LIN {X 0,Y 523.987,Z 450.894,A -85,B 0,C 180,E1 -4780.823,E2 -4780.823} C_VEL
LIN {X 0,Y 524.213,Z 441.663,A -85,B 0,C 180,E1 -4782.19,E2 -4782.19} C_VEL
LIN {X 0,Y 524.572,Z 432.281,A -85,B 0,C 180,E1 -4783.362,E2 -4783.362} C_VEL
LIN {X 0,Y 525.021,Z 420.113,A -85,B 0,C 180,E1 -4784.635,E2 -4784.635} C_VEL
LIN {X 0,Y 525.435,Z 408.795,A -85,B 0,C 180,E1 -4785.626,E2 -4785.626} C_VEL
LIN {X 0,Y 525.945,Z 395.479,A -85,B 0,C 180,E1 -4786.596,E2 -4786.596} C_VEL
LIN {X 0,Y 526.353,Z 382.284,A -85,B 0,C 180,E1 -4787.383,E2 -4787.383} C_VEL
LIN {X 0,Y 526.835,Z 368.983,A -85,B 0,C 180,E1 -4788.018,E2 -4788.018} C_VEL
LIN {X 0,Y 527.198,Z 354.45,A -85,B 0,C 180,E1 -4788.559,E2 -4788.559} C_VEL
LIN {X 0,Y 527.465,Z 339.899,A -85,B 0,C 180,E1 -4788.947,E2 -4788.947} C_VEL
LIN {X 0,Y 527.698,Z 319.361,A -85,B 0,C 180,E1 -4789.281,E2 -4789.281} C_VEL
LIN {X 0,Y 528.518,Z 183.704,A -85,B 0,C 180,E1 -4791.174,E2 -4791.174} C_VEL
LIN {X 0,Y 525.728,Z 169.853,A -85,B 0,C 180,E1 -4791.514,E2 -4791.514} C_VEL
LIN {X 0,Y 526.312,Z 151.353,A -85,B 0,C 180,E1 -4794.034,E2 -4794.034} C_VEL
LIN {X 0,Y 526.522,Z 142.38,A -85,B 0,C 180,E1 -4795.286,E2 -4795.286} C_VEL
LIN {X 0,Y 524.011,Z 130.952,A -85,B 0,C 180,E1 -4797.076,E2 -4797.076} C_VEL
LIN {X 0,Y 523.943,Z 130.846,A -85,B 0,C 180,E1 -4799.756,E2 -4799.756} C_VEL
LIN {X 0,Y 523.934,Z 130.835,A -85,B 0,C 180,E1 -4802.45,E2 -4802.45} C_VEL
LIN {X 0,Y 523.92,Z 130.845,A -85,B 0,C 180,E1 -4805.227,E2 -4805.227} C_VEL
LIN {X 0,Y 523.917,Z 130.849,A -85,B 0,C 180,E1 -4808.102,E2 -4808.102} C_VEL
LIN {X 0,Y 523.939,Z 130.842,A -85,B 0,C 180,E1 -4811.092,E2 -4811.092} C_VEL
LIN {X 0,Y 523.932,Z 130.842,A -85,B 0,C 180,E1 -4814.229,E2 -4814.229} C_VEL
LIN {X 0,Y 523.922,Z 130.844,A -85,B 0,C 180,E1 -4816.833,E2 -4816.833} C_VEL
LIN {X 0,Y 523.938,Z 130.839,A -85,B 0,C 180,E1 -4819.87,E2 -4819.87} C_VEL
LIN {X 0,Y 523.908,Z 130.847,A -85,B 0,C 180,E1 -4822.868,E2 -4822.868} C_VEL
LIN {X 0,Y 523.921,Z 130.836,A -85,B 0,C 180,E1 -4825.709,E2 -4825.709} C_VEL
LIN {X 0,Y 523.92,Z 130.835,A -85,B 0,C 180,E1 -4828.456,E2 -4828.456} C_VEL
LIN {X 0,Y 523.936,Z 130.847,A -85,B 0,C 180,E1 -4831.125,E2 -4831.125} C_VEL
LIN {X 0,Y 523.984,Z 130.833,A -85,B 0,C 180,E1 -4833.981,E2 -4833.981} C_VEL
LIN {X 0,Y 523.925,Z 130.843,A -85,B 0,C 180,E1 -4836.27,E2 -4836.27} C_VEL
LIN {X 0,Y 523.947,Z 130.842,A -85,B 0,C 180,E1 -4838.767,E2 -4838.767} C_VEL
LIN {X 0,Y 523.939,Z 130.847,A -85,B 0,C 180,E1 -4841.22,E2 -4841.22} C_VEL
LIN {X 0,Y 523.923,Z 130.84,A -85,B 0,C 180,E1 -4843.639,E2 -4843.639} C_VEL
LIN {X 0,Y 523.933,Z 130.841,A -85,B 0,C 180,E1 -4846.028,E2 -4846.028} C_VEL
LIN {X 0,Y 524.015,Z 130.835,A -85,B 0,C 180,E1 -4848.394,E2 -4848.394} C_VEL
LIN {X 0,Y 523.989,Z 130.833,A -85,B 0,C 180,E1 -4851.516,E2 -4851.516} C_VEL
LIN {X 0,Y 524.079,Z 130.829,A -85,B 0,C 180,E1 -4854.614,E2 -4854.614} C_VEL
LIN {X 0,Y 524.112,Z 130.817,A -85,B 0,C 180,E1 -4857.695,E2 -4857.695} C_VEL
LIN {X 0,Y 524.122,Z 130.819,A -85,B 0,C 180,E1 -4860.768,E2 -4860.768} C_VEL
LIN {X 0,Y 524.032,Z 130.827,A -85,B 0,C 180,E1 -4863.075,E2 -4863.075} C_VEL
LIN {X 0,Y 524.029,Z 130.837,A -85,B 0,C 180,E1 -4866.159,E2 -4866.159} C_VEL
LIN {X 0,Y 523.987,Z 130.831,A -85,B 0,C 180,E1 -4869.262,E2 -4869.262} C_VEL
LIN {X 0,Y 524.001,Z 130.837,A -85,B 0,C 180,E1 -4871.737,E2 -4871.737} C_VEL
LIN {X 0,Y 523.989,Z 130.831,A -85,B 0,C 180,E1 -4875.049,E2 -4875.049} C_VEL
LIN {X 0,Y 523.916,Z 130.852,A -85,B 0,C 180,E1 -4877.971,E2 -4877.971} C_VEL
LIN {X 0,Y 523.959,Z 130.839,A -85,B 0,C 180,E1 -4880.411,E2 -4880.411} C_VEL
LIN {X 0,Y 523.908,Z 130.845,A -85,B 0,C 180,E1 -4882.894,E2 -4882.894} C_VEL
LIN {X 0,Y 523.901,Z 130.846,A -85,B 0,C 180,E1 -4885.421,E2 -4885.421} C_VEL
LIN {X 0,Y 523.912,Z 130.849,A -85,B 0,C 180,E1 -4888.002,E2 -4888.002} C_VEL
LIN {X 0,Y 523.936,Z 130.835,A -85,B 0,C 180,E1 -4890.853,E2 -4890.853} C_VEL
LIN {X 0,Y 523.927,Z 130.841,A -85,B 0,C 180,E1 -4893.729,E2 -4893.729} C_VEL
LIN {X 0,Y 523.898,Z 130.847,A -85,B 0,C 180,E1 -4896.4,E2 -4896.4} C_VEL
LIN {X 0,Y 523.912,Z 130.845,A -85,B 0,C 180,E1 -4899.086,E2 -4899.086} C_VEL
LIN {X 0,Y 523.899,Z 130.845,A -85,B 0,C 180,E1 -4902.124,E2 -4902.124} C_VEL
LIN {X 0,Y 523.934,Z 130.842,A -85,B 0,C 180,E1 -4905.311,E2 -4905.311} C_VEL
LIN {X 0,Y 523.878,Z 130.847,A -85,B 0,C 180,E1 -4906.896,E2 -4906.896} C_VEL
LIN {X 0,Y 523.2,Z 130.938,A -85,B 0,C 180,E1 -4907.538,E2 -4907.538} C_VEL
LIN {X 0,Y 520.357,Z 131.291,A -85,B 0,C 180,E1 -4908.579,E2 -4908.579} C_VEL
LIN {X 0,Y 517.964,Z 131.586,A -85,B 0,C 180,E1 -4909.418,E2 -4909.418} C_VEL
LIN {X 0,Y 516.94,Z 131.709,A -85,B 0,C 180,E1 -4910.066,E2 -4910.066} C_VEL
LIN {X 0,Y 516.858,Z 131.719,A -85,B 0,C 180,E1 -4910.285,E2 -4910.285} C_VEL
LIN {X 0,Y 516.85,Z 131.726,A -85,B 0,C 180,E1 -4913.252,E2 -4913.252} C_VEL
LIN {X 0,Y 516.879,Z 131.722,A -85,B 0,C 180,E1 -4916.118,E2 -4916.118} C_VEL
LIN {X 0,Y 516.849,Z 131.72,A -85,B 0,C 180,E1 -4918.944,E2 -4918.944} C_VEL
LIN {X 0,Y 516.856,Z 131.728,A -85,B 0,C 180,E1 -4922.11,E2 -4922.11} C_VEL
LIN {X 0,Y 516.864,Z 131.779,A -85,B 0,C 180,E1 -4923.695,E2 -4923.695} C_VEL
LIN {X 0,Y 517.122,Z 133.046,A -85,B 0,C 180,E1 -4923.969,E2 -4923.969} C_VEL
LIN {X 0,Y 519.393,Z 143.168,A -85,B 0,C 180,E1 -4925.625,E2 -4925.625} C_VEL
LIN {X 0,Y 519.177,Z 153.314,A -85,B 0,C 180,E1 -4927.13,E2 -4927.13} C_VEL
LIN {X 0,Y 518.951,Z 161.322,A -85,B 0,C 180,E1 -4928.255,E2 -4928.255} C_VEL
LIN {X 0,Y 521.967,Z 176.108,A -85,B 0,C 180,E1 -4928.615,E2 -4928.615} C_VEL
LIN {X 0,Y 520.906,Z 326.105,A -85,B 0,C 180,E1 -4930.75,E2 -4930.75} C_VEL
LIN {X 0,Y 520.589,Z 341.471,A -85,B 0,C 180,E1 -4931.12,E2 -4931.12} C_VEL
LIN {X 0,Y 520.263,Z 356.352,A -85,B 0,C 180,E1 -4931.644,E2 -4931.644} C_VEL
LIN {X 0,Y 519.75,Z 370.274,A -85,B 0,C 180,E1 -4932.287,E2 -4932.287} C_VEL
LIN {X 0,Y 519.241,Z 383.909,A -85,B 0,C 180,E1 -4933.082,E2 -4933.082} C_VEL
LIN {X 0,Y 518.727,Z 396.578,A -85,B 0,C 180,E1 -4933.986,E2 -4933.986} C_VEL
LIN {X 0,Y 518.184,Z 409.14,A -85,B 0,C 180,E1 -4935.067,E2 -4935.067} C_VEL
LIN {X 0,Y 517.708,Z 420.65,A -85,B 0,C 180,E1 -4936.257,E2 -4936.257} C_VEL
LIN {X 0,Y 517.314,Z 430.339,A -85,B 0,C 180,E1 -4937.445,E2 -4937.445} C_VEL
LIN {X 0,Y 517.023,Z 439.835,A -85,B 0,C 180,E1 -4938.831,E2 -4938.831} C_VEL
LIN {X 0,Y 516.725,Z 447.744,A -85,B 0,C 180,E1 -4940.211,E2 -4940.211} C_VEL
LIN {X 0,Y 516.511,Z 455.13,A -85,B 0,C 180,E1 -4941.786,E2 -4941.786} C_VEL
LIN {X 0,Y 516.394,Z 459.661,A -85,B 0,C 180,E1 -4942.964,E2 -4942.964} C_VEL
LIN {X 0,Y 516.379,Z 464.465,A -85,B 0,C 180,E1 -4944.533,E2 -4944.533} C_VEL
LIN {X 0,Y 516.307,Z 467.988,A -85,B 0,C 180,E1 -4946.097,E2 -4946.097} C_VEL
LIN {X 0,Y 516.259,Z 470.322,A -85,B 0,C 180,E1 -4947.659,E2 -4947.659} C_VEL
LIN {X 0,Y 516.156,Z 471.518,A -85,B 0,C 180,E1 -4949.22,E2 -4949.22} C_VEL
LIN {X 0,Y 516.157,Z 471.537,A -85,B 0,C 180,E1 -4950.78,E2 -4950.78} C_VEL
LIN {X 0,Y 516.259,Z 470.418,A -85,B 0,C 180,E1 -4952.341,E2 -4952.341} C_VEL
LIN {X 0,Y 516.308,Z 468.16,A -85,B 0,C 180,E1 -4953.903,E2 -4953.903} C_VEL
LIN {X 0,Y 516.374,Z 464.708,A -85,B 0,C 180,E1 -4955.467,E2 -4955.467} C_VEL
LIN {X 0,Y 516.393,Z 459.982,A -85,B 0,C 180,E1 -4957.036,E2 -4957.036} C_VEL
LIN {X 0,Y 516.542,Z 453.859,A -85,B 0,C 180,E1 -4958.608,E2 -4958.608} C_VEL
LIN {X 0,Y 516.767,Z 446.151,A -85,B 0,C 180,E1 -4960.183,E2 -4960.183} C_VEL
LIN {X 0,Y 517.008,Z 437.932,A -85,B 0,C 180,E1 -4961.567,E2 -4961.567} C_VEL
LIN {X 0,Y 517.394,Z 428.037,A -85,B 0,C 180,E1 -4962.952,E2 -4962.952} C_VEL
LIN {X 0,Y 517.838,Z 417.892,A -85,B 0,C 180,E1 -4964.14,E2 -4964.14} C_VEL
LIN {X 0,Y 518.342,Z 406.115,A -85,B 0,C 180,E1 -4965.303,E2 -4965.303} C_VEL
LIN {X 0,Y 518.84,Z 393.976,A -85,B 0,C 180,E1 -4966.304,E2 -4966.304} C_VEL
LIN {X 0,Y 519.399,Z 380.576,A -85,B 0,C 180,E1 -4967.217,E2 -4967.217} C_VEL
LIN {X 0,Y 519.804,Z 368.066,A -85,B 0,C 180,E1 -4967.914,E2 -4967.914} C_VEL
LIN {X 0,Y 520.338,Z 353.435,A -85,B 0,C 180,E1 -4968.557,E2 -4968.557} C_VEL
LIN {X 0,Y 520.652,Z 338.696,A -85,B 0,C 180,E1 -4969.044,E2 -4969.044} C_VEL
LIN {X 0,Y 520.941,Z 323.655,A -85,B 0,C 180,E1 -4969.38,E2 -4969.38} C_VEL
LIN {X 0,Y 522.001,Z 175.538,A -85,B 0,C 180,E1 -4971.482,E2 -4971.482} C_VEL
LIN {X 0,Y 518.92,Z 161.155,A -85,B 0,C 180,E1 -4971.846,E2 -4971.846} C_VEL
LIN {X 0,Y 519.489,Z 145.188,A -85,B 0,C 180,E1 -4974.157,E2 -4974.157} C_VEL
LIN {X 0,Y 518.911,Z 140.798,A -85,B 0,C 180,E1 -4974.847,E2 -4974.847} C_VEL
LIN {X 0,Y 516.893,Z 132.05,A -85,B 0,C 180,E1 -4976.307,E2 -4976.307} C_VEL
LIN {X 0,Y 516.828,Z 131.719,A -85,B 0,C 180,E1 -4976.663,E2 -4976.663} C_VEL
LIN {X 0,Y 516.838,Z 131.719,A -85,B 0,C 180,E1 -4979.509,E2 -4979.509} C_VEL
LIN {X 0,Y 516.867,Z 131.726,A -85,B 0,C 180,E1 -4982.538,E2 -4982.538} C_VEL
LIN {X 0,Y 516.851,Z 131.729,A -85,B 0,C 180,E1 -4985.327,E2 -4985.327} C_VEL
LIN {X 0,Y 516.869,Z 131.728,A -85,B 0,C 180,E1 -4988.717,E2 -4988.717} C_VEL
LIN {X 0,Y 516.845,Z 131.726,A -85,B 0,C 180,E1 -4991.782,E2 -4991.782} C_VEL
LIN {X 0,Y 516.897,Z 131.722,A -85,B 0,C 180,E1 -4995.007,E2 -4995.007} C_VEL
LIN {X 0,Y 516.85,Z 131.728,A -85,B 0,C 180,E1 -4998.407,E2 -4998.407} C_VEL
LIN {X 0,Y 516.875,Z 131.719,A -85,B 0,C 180,E1 -5001.283,E2 -5001.283} C_VEL
LIN {X 0,Y 516.866,Z 131.727,A -85,B 0,C 180,E1 -5004.219,E2 -5004.219} C_VEL
LIN {X 0,Y 516.882,Z 131.707,A -85,B 0,C 180,E1 -5007.052,E2 -5007.052} C_VEL
LIN {X 0,Y 516.866,Z 131.715,A -85,B 0,C 180,E1 -5009.795,E2 -5009.795} C_VEL
LIN {X 0,Y 516.876,Z 131.728,A -85,B 0,C 180,E1 -5012.464,E2 -5012.464} C_VEL
LIN {X 0,Y 516.847,Z 131.721,A -85,B 0,C 180,E1 -5015.068,E2 -5015.068} C_VEL
LIN {X 0,Y 516.871,Z 131.724,A -85,B 0,C 180,E1 -5017.622,E2 -5017.622} C_VEL
LIN {X 0,Y 516.92,Z 131.718,A -85,B 0,C 180,E1 -5020.129,E2 -5020.129} C_VEL
LIN {X 0,Y 516.881,Z 131.723,A -85,B 0,C 180,E1 -5022.594,E2 -5022.594} C_VEL
LIN {X 0,Y 516.938,Z 131.709,A -85,B 0,C 180,E1 -5025.03,E2 -5025.03} C_VEL
LIN {X 0,Y 516.969,Z 131.714,A -85,B 0,C 180,E1 -5028.234,E2 -5028.234} C_VEL
LIN {X 0,Y 516.955,Z 131.711,A -85,B 0,C 180,E1 -5031.399,E2 -5031.399} C_VEL
LIN {X 0,Y 517.022,Z 131.703,A -85,B 0,C 180,E1 -5034.54,E2 -5034.54} C_VEL
LIN {X 0,Y 517.081,Z 131.696,A -85,B 0,C 180,E1 -5037.663,E2 -5037.663} C_VEL
LIN {X 0,Y 517.088,Z 131.697,A -85,B 0,C 180,E1 -5040,E2 -5040} C_VEL
LIN {X 0,Y 517.082,Z 131.692,A -85,B 0,C 180,E1 -5042.337,E2 -5042.337} C_VEL
LIN {X 0,Y 517.025,Z 131.708,A -85,B 0,C 180,E1 -5045.46,E2 -5045.46} C_VEL
LIN {X 0,Y 516.957,Z 131.709,A -85,B 0,C 180,E1 -5048.6,E2 -5048.6} C_VEL
LIN {X 0,Y 516.954,Z 131.713,A -85,B 0,C 180,E1 -5051.807,E2 -5051.807} C_VEL
LIN {X 0,Y 516.945,Z 131.714,A -85,B 0,C 180,E1 -5055.145,E2 -5055.145} C_VEL
LIN {X 0,Y 516.914,Z 131.717,A -85,B 0,C 180,E1 -5058.223,E2 -5058.223} C_VEL
LIN {X 0,Y 516.914,Z 131.719,A -85,B 0,C 180,E1 -5060.701,E2 -5060.701} C_VEL
LIN {X 0,Y 516.887,Z 131.72,A -85,B 0,C 180,E1 -5064.073,E2 -5064.073} C_VEL
LIN {X 0,Y 516.91,Z 131.719,A -85,B 0,C 180,E1 -5066.659,E2 -5066.659} C_VEL
LIN {X 0,Y 516.911,Z 131.716,A -85,B 0,C 180,E1 -5069.523,E2 -5069.523} C_VEL
LIN {X 0,Y 516.895,Z 131.708,A -85,B 0,C 180,E1 -5072.543,E2 -5072.543} C_VEL
LIN {X 0,Y 516.867,Z 131.721,A -85,B 0,C 180,E1 -5075.329,E2 -5075.329} C_VEL
LIN {X 0,Y 516.881,Z 131.723,A -85,B 0,C 180,E1 -5077.943,E2 -5077.943} C_VEL
LIN {X 0,Y 516.884,Z 131.717,A -85,B 0,C 180,E1 -5080.742,E2 -5080.742} C_VEL
LIN {X 0,Y 516.885,Z 131.723,A -85,B 0,C 180,E1 -5082.831,E2 -5082.831} C_VEL
LIN {X 0,Y 516.896,Z 131.715,A -85,B 0,C 180,E1 -5085.007,E2 -5085.007} C_VEL
LIN {X 0,Y 516.914,Z 131.722,A -85,B 0,C 180,E1 -5088.399,E2 -5088.399} C_VEL
LIN {X 0,Y 516.883,Z 131.719,A -85,B 0,C 180,E1 -5091.284,E2 -5091.284} C_VEL
LIN {X 0,Y 516.872,Z 131.724,A -85,B 0,C 180,E1 -5094.22,E2 -5094.22} C_VEL
LIN {X 0,Y 516.895,Z 131.715,A -85,B 0,C 180,E1 -5097.053,E2 -5097.053} C_VEL
LIN {X 0,Y 516.893,Z 131.723,A -85,B 0,C 180,E1 -5099.796,E2 -5099.796} C_VEL
LIN {X 0,Y 516.941,Z 131.828,A -85,B 0,C 180,E1 -5102.66,E2 -5102.66} C_VEL
LIN {X 0,Y 519.647,Z 143.76,A -85,B 0,C 180,E1 -5104.562,E2 -5104.562} C_VEL
LIN {X 0,Y 519.417,Z 154.273,A -85,B 0,C 180,E1 -5106.051,E2 -5106.051} C_VEL
LIN {X 0,Y 518.893,Z 169.735,A -85,B 0,C 180,E1 -5108.185,E2 -5108.185} C_VEL
LIN {X 0,Y 521.944,Z 185.319,A -85,B 0,C 180,E1 -5108.571,E2 -5108.571} C_VEL
LIN {X 0,Y 520.888,Z 335.251,A -85,B 0,C 180,E1 -5110.704,E2 -5110.704} C_VEL
LIN {X 0,Y 520.559,Z 350.405,A -85,B 0,C 180,E1 -5111.067,E2 -5111.067} C_VEL
LIN {X 0,Y 520.171,Z 365.412,A -85,B 0,C 180,E1 -5111.59,E2 -5111.59} C_VEL
LIN {X 0,Y 519.646,Z 380.411,A -85,B 0,C 180,E1 -5112.284,E2 -5112.284} C_VEL
LIN {X 0,Y 519.132,Z 393.896,A -85,B 0,C 180,E1 -5113.078,E2 -5113.078} C_VEL
LIN {X 0,Y 518.614,Z 407.626,A -85,B 0,C 180,E1 -5114.073,E2 -5114.073} C_VEL
LIN {X 0,Y 518.057,Z 420.039,A -85,B 0,C 180,E1 -5115.164,E2 -5115.164} C_VEL
LIN {X 0,Y 517.593,Z 432.215,A -85,B 0,C 180,E1 -5116.454,E2 -5116.454} C_VEL
LIN {X 0,Y 517.146,Z 443.038,A -85,B 0,C 180,E1 -5117.84,E2 -5117.84} C_VEL
LIN {X 0,Y 516.895,Z 452.046,A -85,B 0,C 180,E1 -5119.225,E2 -5119.225} C_VEL
LIN {X 0,Y 516.601,Z 459.516,A -85,B 0,C 180,E1 -5120.604,E2 -5120.604} C_VEL
LIN {X 0,Y 516.451,Z 466.485,A -85,B 0,C 180,E1 -5122.179,E2 -5122.179} C_VEL
LIN {X 0,Y 516.36,Z 471.963,A -85,B 0,C 180,E1 -5123.749,E2 -5123.749} C_VEL
LIN {X 0,Y 516.239,Z 476.102,A -85,B 0,C 180,E1 -5125.315,E2 -5125.315} C_VEL
LIN {X 0,Y 516.27,Z 479.005,A -85,B 0,C 180,E1 -5126.879,E2 -5126.879} C_VEL
LIN {X 0,Y 516.189,Z 480.735,A -85,B 0,C 180,E1 -5128.44,E2 -5128.44} C_VEL
LIN {X 0,Y 516.151,Z 481.328,A -85,B 0,C 180,E1 -5130,E2 -5130} C_VEL
LIN {X 0,Y 516.189,Z 480.733,A -85,B 0,C 180,E1 -5131.56,E2 -5131.56} C_VEL
LIN {X 0,Y 516.27,Z 479,A -85,B 0,C 180,E1 -5133.121,E2 -5133.121} C_VEL
LIN {X 0,Y 516.239,Z 476.1,A -85,B 0,C 180,E1 -5134.685,E2 -5134.685} C_VEL
LIN {X 0,Y 516.376,Z 471.967,A -85,B 0,C 180,E1 -5136.251,E2 -5136.251} C_VEL
LIN {X 0,Y 516.451,Z 466.486,A -85,B 0,C 180,E1 -5137.821,E2 -5137.821} C_VEL
LIN {X 0,Y 516.601,Z 459.51,A -85,B 0,C 180,E1 -5139.396,E2 -5139.396} C_VEL
LIN {X 0,Y 516.952,Z 450.827,A -85,B 0,C 180,E1 -5140.972,E2 -5140.972} C_VEL
LIN {X 0,Y 517.202,Z 441.748,A -85,B 0,C 180,E1 -5142.338,E2 -5142.338} C_VEL
LIN {X 0,Y 517.593,Z 432.214,A -85,B 0,C 180,E1 -5143.546,E2 -5143.546} C_VEL
LIN {X 0,Y 518.092,Z 420.046,A -85,B 0,C 180,E1 -5144.835,E2 -5144.835} C_VEL
LIN {X 0,Y 518.59,Z 407.889,A -85,B 0,C 180,E1 -5145.908,E2 -5145.908} C_VEL
LIN {X 0,Y 519.082,Z 395.412,A -85,B 0,C 180,E1 -5146.822,E2 -5146.822} C_VEL
LIN {X 0,Y 519.543,Z 382.217,A -85,B 0,C 180,E1 -5147.618,E2 -5147.618} C_VEL
LIN {X 0,Y 520.123,Z 367.788,A -85,B 0,C 180,E1 -5148.31,E2 -5148.31} C_VEL
LIN {X 0,Y 520.471,Z 353.62,A -85,B 0,C 180,E1 -5148.833,E2 -5148.833} C_VEL
LIN {X 0,Y 520.812,Z 338.587,A -85,B 0,C 180,E1 -5149.227,E2 -5149.227} C_VEL
LIN {X 0,Y 521.012,Z 316.274,A -85,B 0,C 180,E1 -5149.582,E2 -5149.582} C_VEL
LIN {X 0,Y 521.92,Z 184.769,A -85,B 0,C 180,E1 -5151.438,E2 -5151.438} C_VEL
LIN {X 0,Y 518.869,Z 169.838,A -85,B 0,C 180,E1 -5151.809,E2 -5151.809} C_VEL
LIN {X 0,Y 519.47,Z 152.785,A -85,B 0,C 180,E1 -5154.158,E2 -5154.158} C_VEL
LIN {X 0,Y 519.759,Z 144.939,A -85,B 0,C 180,E1 -5155.263,E2 -5155.263} C_VEL
LIN {X 0,Y 517.664,Z 134.82,A -85,B 0,C 180,E1 -5156.834,E2 -5156.834} C_VEL
LIN {X 0,Y 516.957,Z 131.788,A -85,B 0,C 180,E1 -5157.366,E2 -5157.366} C_VEL
LIN {X 0,Y 516.893,Z 131.723,A -85,B 0,C 180,E1 -5160.204,E2 -5160.204} C_VEL
LIN {X 0,Y 516.895,Z 131.716,A -85,B 0,C 180,E1 -5162.947,E2 -5162.947} C_VEL
LIN {X 0,Y 516.871,Z 131.724,A -85,B 0,C 180,E1 -5165.78,E2 -5165.78} C_VEL
LIN {X 0,Y 516.883,Z 131.718,A -85,B 0,C 180,E1 -5168.716,E2 -5168.716} C_VEL
LIN {X 0,Y 516.912,Z 131.725,A -85,B 0,C 180,E1 -5171.775,E2 -5171.775} C_VEL
LIN {X 0,Y 516.895,Z 131.716,A -85,B 0,C 180,E1 -5175.007,E2 -5175.007} C_VEL
LIN {X 0,Y 516.914,Z 131.711,A -85,B 0,C 180,E1 -5178.399,E2 -5178.399} C_VEL
LIN {X 0,Y 516.881,Z 131.719,A -85,B 0,C 180,E1 -5181.284,E2 -5181.284} C_VEL
LIN {X 0,Y 516.872,Z 131.72,A -85,B 0,C 180,E1 -5184.22,E2 -5184.22} C_VEL
LIN {X 0,Y 516.882,Z 131.708,A -85,B 0,C 180,E1 -5187.052,E2 -5187.052} C_VEL
LIN {X 0,Y 516.888,Z 131.722,A -85,B 0,C 180,E1 -5189.796,E2 -5189.796} C_VEL
LIN {X 0,Y 516.926,Z 131.715,A -85,B 0,C 180,E1 -5192.467,E2 -5192.467} C_VEL
LIN {X 0,Y 516.907,Z 131.72,A -85,B 0,C 180,E1 -5195.072,E2 -5195.072} C_VEL
LIN {X 0,Y 516.887,Z 131.718,A -85,B 0,C 180,E1 -5198.462,E2 -5198.462} C_VEL
LIN {X 0,Y 516.893,Z 131.725,A -85,B 0,C 180,E1 -5200.955,E2 -5200.955} C_VEL
LIN {X 0,Y 516.899,Z 131.717,A -85,B 0,C 180,E1 -5203.41,E2 -5203.41} C_VEL
LIN {X 0,Y 516.889,Z 131.718,A -85,B 0,C 180,E1 -5205.834,E2 -5205.834} C_VEL
LIN {X 0,Y 516.952,Z 131.713,A -85,B 0,C 180,E1 -5209.028,E2 -5209.028} C_VEL
LIN {X 0,Y 516.964,Z 131.71,A -85,B 0,C 180,E1 -5212.187,E2 -5212.187} C_VEL
LIN {X 0,Y 517.026,Z 131.709,A -85,B 0,C 180,E1 -5214.54,E2 -5214.54} C_VEL
LIN {X 0,Y 517.083,Z 131.692,A -85,B 0,C 180,E1 -5217.663,E2 -5217.663} C_VEL
LIN {X 0,Y 517.092,Z 131.695,A -85,B 0,C 180,E1 -5220.779,E2 -5220.779} C_VEL
LIN {X 0,Y 516.974,Z 131.706,A -85,B 0,C 180,E1 -5223.117,E2 -5223.117} C_VEL
LIN {X 0,Y 516.991,Z 131.715,A -85,B 0,C 180,E1 -5226.243,E2 -5226.243} C_VEL
LIN {X 0,Y 516.943,Z 131.709,A -85,B 0,C 180,E1 -5229.39,E2 -5229.39} C_VEL
LIN {X 0,Y 516.954,Z 131.715,A -85,B 0,C 180,E1 -5231.807,E2 -5231.807} C_VEL
LIN {X 0,Y 516.941,Z 131.709,A -85,B 0,C 180,E1 -5235.144,E2 -5235.144} C_VEL
LIN {X 0,Y 516.879,Z 131.724,A -85,B 0,C 180,E1 -5238.224,E2 -5238.224} C_VEL
LIN {X 0,Y 516.906,Z 131.715,A -85,B 0,C 180,E1 -5240.702,E2 -5240.702} C_VEL
LIN {X 0,Y 516.886,Z 131.721,A -85,B 0,C 180,E1 -5244.073,E2 -5244.073} C_VEL
LIN {X 0,Y 516.845,Z 131.725,A -85,B 0,C 180,E1 -5246.662,E2 -5246.662} C_VEL
LIN {X 0,Y 516.887,Z 131.724,A -85,B 0,C 180,E1 -5249.519,E2 -5249.519} C_VEL
LIN {X 0,Y 516.895,Z 131.703,A -85,B 0,C 180,E1 -5252.543,E2 -5252.543} C_VEL
LIN {X 0,Y 516.861,Z 131.726,A -85,B 0,C 180,E1 -5255.329,E2 -5255.329} C_VEL
LIN {X 0,Y 516.878,Z 131.719,A -85,B 0,C 180,E1 -5257.942,E2 -5257.942} C_VEL
LIN {X 0,Y 516.853,Z 131.712,A -85,B 0,C 180,E1 -5260.745,E2 -5260.745} C_VEL
LIN {X 0,Y 516.881,Z 131.722,A -85,B 0,C 180,E1 -5263.904,E2 -5263.904} C_VEL
LIN {X 0,Y 516.836,Z 131.725,A -85,B 0,C 180,E1 -5266.896,E2 -5266.896} C_VEL
LIN {X 0,Y 516.86,Z 131.721,A -85,B 0,C 180,E1 -5269.593,E2 -5269.593} C_VEL
LIN {X 0,Y 516.858,Z 131.719,A -85,B 0,C 180,E1 -5270.285,E2 -5270.285} C_VEL
LIN {X 0,Y 516.197,Z 131.809,A -85,B 0,C 180,E1 -5270.936,E2 -5270.936} C_VEL
LIN {X 0,Y 513.348,Z 132.162,A -85,B 0,C 180,E1 -5271.991,E2 -5271.991} C_VEL
LIN {X 0,Y 510.932,Z 132.468,A -85,B 0,C 180,E1 -5272.842,E2 -5272.842} C_VEL
LIN {X 0,Y 509.888,Z 132.593,A -85,B 0,C 180,E1 -5273.498,E2 -5273.498} C_VEL
LIN {X 0,Y 509.8,Z 132.602,A -85,B 0,C 180,E1 -5273.721,E2 -5273.721} C_VEL
LIN {X 0,Y 509.839,Z 132.6,A -85,B 0,C 180,E1 -5276.538,E2 -5276.538} C_VEL
LIN {X 0,Y 509.801,Z 132.592,A -85,B 0,C 180,E1 -5279.331,E2 -5279.331} C_VEL
LIN {X 0,Y 509.823,Z 132.604,A -85,B 0,C 180,E1 -5282.05,E2 -5282.05} C_VEL
LIN {X 0,Y 509.803,Z 132.654,A -85,B 0,C 180,E1 -5283.429,E2 -5283.429} C_VEL
LIN {X 0,Y 510.265,Z 134.76,A -85,B 0,C 180,E1 -5283.849,E2 -5283.849} C_VEL
LIN {X 0,Y 512.569,Z 144.901,A -85,B 0,C 180,E1 -5285.534,E2 -5285.534} C_VEL
LIN {X 0,Y 512.234,Z 156.336,A -85,B 0,C 180,E1 -5287.247,E2 -5287.247} C_VEL
LIN {X 0,Y 512.117,Z 161.303,A -85,B 0,C 180,E1 -5287.944,E2 -5287.944} C_VEL
LIN {X 0,Y 515.308,Z 176.214,A -85,B 0,C 180,E1 -5288.324,E2 -5288.324} C_VEL
LIN {X 0,Y 514.261,Z 322.379,A -85,B 0,C 180,E1 -5290.425,E2 -5290.425} C_VEL
LIN {X 0,Y 513.998,Z 337.997,A -85,B 0,C 180,E1 -5290.768,E2 -5290.768} C_VEL
LIN {X 0,Y 513.616,Z 352.541,A -85,B 0,C 180,E1 -5291.243,E2 -5291.243} C_VEL
LIN {X 0,Y 513.103,Z 366.388,A -85,B 0,C 180,E1 -5291.844,E2 -5291.844} C_VEL
LIN {X 0,Y 512.555,Z 380.825,A -85,B 0,C 180,E1 -5292.649,E2 -5292.649} C_VEL
LIN {X 0,Y 511.971,Z 393.945,A -85,B 0,C 180,E1 -5293.553,E2 -5293.553} C_VEL
LIN {X 0,Y 511.488,Z 405.439,A -85,B 0,C 180,E1 -5294.506,E2 -5294.506} C_VEL
LIN {X 0,Y 510.948,Z 417.161,A -85,B 0,C 180,E1 -5295.665,E2 -5295.665} C_VEL
LIN {X 0,Y 510.48,Z 427.389,A -85,B 0,C 180,E1 -5296.87,E2 -5296.87} C_VEL
LIN {X 0,Y 510.051,Z 436.916,A -85,B 0,C 180,E1 -5298.201,E2 -5298.201} C_VEL
LIN {X 0,Y 509.832,Z 444.596,A -85,B 0,C 180,E1 -5299.476,E2 -5299.476} C_VEL
LIN {X 0,Y 509.551,Z 451.709,A -85,B 0,C 180,E1 -5300.874,E2 -5300.874} C_VEL
LIN {X 0,Y 509.355,Z 458.31,A -85,B 0,C 180,E1 -5302.468,E2 -5302.468} C_VEL
LIN {X 0,Y 509.304,Z 463.473,A -85,B 0,C 180,E1 -5304.06,E2 -5304.06} C_VEL
LIN {X 0,Y 509.16,Z 466.449,A -85,B 0,C 180,E1 -5305.249,E2 -5305.249} C_VEL
LIN {X 0,Y 509.188,Z 469.367,A -85,B 0,C 180,E1 -5306.835,E2 -5306.835} C_VEL
LIN {X 0,Y 509.11,Z 471.127,A -85,B 0,C 180,E1 -5308.418,E2 -5308.418} C_VEL
LIN {X 0,Y 509.064,Z 471.744,A -85,B 0,C 180,E1 -5310,E2 -5310} C_VEL
LIN {X 0,Y 509.111,Z 471.184,A -85,B 0,C 180,E1 -5311.582,E2 -5311.582} C_VEL
LIN {X 0,Y 509.189,Z 469.499,A -85,B 0,C 180,E1 -5313.165,E2 -5313.165} C_VEL
LIN {X 0,Y 509.159,Z 466.653,A -85,B 0,C 180,E1 -5314.751,E2 -5314.751} C_VEL
LIN {X 0,Y 509.287,Z 463.71,A -85,B 0,C 180,E1 -5315.941,E2 -5315.941} C_VEL
LIN {X 0,Y 509.354,Z 458.628,A -85,B 0,C 180,E1 -5317.532,E2 -5317.532} C_VEL
LIN {X 0,Y 509.544,Z 452.12,A -85,B 0,C 180,E1 -5319.127,E2 -5319.127} C_VEL
LIN {X 0,Y 509.828,Z 445.1,A -85,B 0,C 180,E1 -5320.524,E2 -5320.524} C_VEL
LIN {X 0,Y 510.081,Z 436.366,A -85,B 0,C 180,E1 -5321.971,E2 -5321.971} C_VEL
LIN {X 0,Y 510.517,Z 426.486,A -85,B 0,C 180,E1 -5323.332,E2 -5323.332} C_VEL
LIN {X 0,Y 510.979,Z 416.088,A -85,B 0,C 180,E1 -5324.537,E2 -5324.537} C_VEL
LIN {X 0,Y 511.524,Z 404.997,A -85,B 0,C 180,E1 -5325.623,E2 -5325.623} C_VEL
LIN {X 0,Y 512.062,Z 392.484,A -85,B 0,C 180,E1 -5326.649,E2 -5326.649} C_VEL
LIN {X 0,Y 512.666,Z 379.052,A -85,B 0,C 180,E1 -5327.553,E2 -5327.553} C_VEL
LIN {X 0,Y 513.217,Z 364.109,A -85,B 0,C 180,E1 -5328.359,E2 -5328.359} C_VEL
LIN {X 0,Y 513.736,Z 348.826,A -85,B 0,C 180,E1 -5328.986,E2 -5328.986} C_VEL
LIN {X 0,Y 514.063,Z 333.893,A -85,B 0,C 180,E1 -5329.433,E2 -5329.433} C_VEL
LIN {X 0,Y 514.312,Z 319.15,A -85,B 0,C 180,E1 -5329.718,E2 -5329.718} C_VEL
LIN {X 0,Y 515.386,Z 176.758,A -85,B 0,C 180,E1 -5331.754,E2 -5331.754} C_VEL
LIN {X 0,Y 512.116,Z 161.267,A -85,B 0,C 180,E1 -5332.149,E2 -5332.149} C_VEL
LIN {X 0,Y 512.657,Z 145.463,A -85,B 0,C 180,E1 -5334.467,E2 -5334.467} C_VEL
LIN {X 0,Y 509.843,Z 132.917,A -85,B 0,C 180,E1 -5336.573,E2 -5336.573} C_VEL
LIN {X 0,Y 509.782,Z 132.595,A -85,B 0,C 180,E1 -5336.771,E2 -5336.771} C_VEL
LIN {X 0,Y 509.793,Z 132.609,A -85,B 0,C 180,E1 -5338.85,E2 -5338.85} C_VEL
LIN {X 0,Y 509.789,Z 132.608,A -85,B 0,C 180,E1 -5341.592,E2 -5341.592} C_VEL
LIN {X 0,Y 509.833,Z 132.599,A -85,B 0,C 180,E1 -5344.415,E2 -5344.415} C_VEL
LIN {X 0,Y 509.783,Z 132.611,A -85,B 0,C 180,E1 -5347.344,E2 -5347.344} C_VEL
LIN {X 0,Y 509.813,Z 132.597,A -85,B 0,C 180,E1 -5350.385,E2 -5350.385} C_VEL
LIN {X 0,Y 509.806,Z 132.597,A -85,B 0,C 180,E1 -5353.573,E2 -5353.573} C_VEL
LIN {X 0,Y 509.806,Z 132.605,A -85,B 0,C 180,E1 -5356.427,E2 -5356.427} C_VEL
LIN {X 0,Y 509.813,Z 132.588,A -85,B 0,C 180,E1 -5359.615,E2 -5359.615} C_VEL
LIN {X 0,Y 509.808,Z 132.607,A -85,B 0,C 180,E1 -5362.658,E2 -5362.658} C_VEL
LIN {X 0,Y 509.84,Z 132.595,A -85,B 0,C 180,E1 -5365.801,E2 -5365.801} C_VEL
LIN {X 0,Y 509.845,Z 132.588,A -85,B 0,C 180,E1 -5368.721,E2 -5368.721} C_VEL
LIN {X 0,Y 509.838,Z 132.598,A -85,B 0,C 180,E1 -5371.153,E2 -5371.153} C_VEL
LIN {X 0,Y 509.851,Z 132.598,A -85,B 0,C 180,E1 -5373.826,E2 -5373.826} C_VEL
LIN {X 0,Y 509.82,Z 132.606,A -85,B 0,C 180,E1 -5376.436,E2 -5376.436} C_VEL
LIN {X 0,Y 509.908,Z 132.591,A -85,B 0,C 180,E1 -5379.844,E2 -5379.844} C_VEL
LIN {X 0,Y 509.854,Z 132.601,A -85,B 0,C 180,E1 -5382.347,E2 -5382.347} C_VEL
LIN {X 0,Y 509.888,Z 132.588,A -85,B 0,C 180,E1 -5384.818,E2 -5384.818} C_VEL
LIN {X 0,Y 509.904,Z 132.595,A -85,B 0,C 180,E1 -5388.124,E2 -5388.124} C_VEL
LIN {X 0,Y 509.903,Z 132.587,A -85,B 0,C 180,E1 -5391.279,E2 -5391.279} C_VEL
LIN {X 0,Y 509.973,Z 132.582,A -85,B 0,C 180,E1 -5394.464,E2 -5394.464} C_VEL
LIN {X 0,Y 510.051,Z 132.571,A -85,B 0,C 180,E1 -5397.631,E2 -5397.631} C_VEL
LIN {X 0,Y 510.02,Z 132.575,A -85,B 0,C 180,E1 -5400.789,E2 -5400.789} C_VEL
LIN {X 0,Y 509.927,Z 132.588,A -85,B 0,C 180,E1 -5403.16,E2 -5403.16} C_VEL
LIN {X 0,Y 509.943,Z 132.584,A -85,B 0,C 180,E1 -5406.33,E2 -5406.33} C_VEL
LIN {X 0,Y 509.905,Z 132.589,A -85,B 0,C 180,E1 -5408.72,E2 -5408.72} C_VEL
LIN {X 0,Y 509.907,Z 132.59,A -85,B 0,C 180,E1 -5411.932,E2 -5411.932} C_VEL
LIN {X 0,Y 509.897,Z 132.591,A -85,B 0,C 180,E1 -5415.242,E2 -5415.242} C_VEL
LIN {X 0,Y 509.859,Z 132.598,A -85,B 0,C 180,E1 -5418.484,E2 -5418.484} C_VEL
LIN {X 0,Y 509.852,Z 132.598,A -85,B 0,C 180,E1 -5421.002,E2 -5421.002} C_VEL
LIN {X 0,Y 509.821,Z 132.601,A -85,B 0,C 180,E1 -5423.564,E2 -5423.564} C_VEL
LIN {X 0,Y 509.888,Z 132.59,A -85,B 0,C 180,E1 -5426.372,E2 -5426.372} C_VEL
LIN {X 0,Y 509.876,Z 132.599,A -85,B 0,C 180,E1 -5428.844,E2 -5428.844} C_VEL
LIN {X 0,Y 509.82,Z 132.59,A -85,B 0,C 180,E1 -5431.59,E2 -5431.59} C_VEL
LIN {X 0,Y 509.839,Z 132.59,A -85,B 0,C 180,E1 -5434.414,E2 -5434.414} C_VEL
LIN {X 0,Y 509.818,Z 132.601,A -85,B 0,C 180,E1 -5437.341,E2 -5437.341} C_VEL
LIN {X 0,Y 509.839,Z 132.592,A -85,B 0,C 180,E1 -5440.382,E2 -5440.382} C_VEL
LIN {X 0,Y 509.825,Z 132.601,A -85,B 0,C 180,E1 -5443.062,E2 -5443.062} C_VEL
LIN {X 0,Y 509.823,Z 132.598,A -85,B 0,C 180,E1 -5445.793,E2 -5445.793} C_VEL
LIN {X 0,Y 509.856,Z 132.599,A -85,B 0,C 180,E1 -5448.574,E2 -5448.574} C_VEL
LIN {X 0,Y 509.852,Z 132.599,A -85,B 0,C 180,E1 -5451.786,E2 -5451.786} C_VEL
LIN {X 0,Y 509.831,Z 132.602,A -85,B 0,C 180,E1 -5454.622,E2 -5454.622} C_VEL
LIN {X 0,Y 509.862,Z 132.585,A -85,B 0,C 180,E1 -5457.481,E2 -5457.481} C_VEL
LIN {X 0,Y 509.859,Z 132.601,A -85,B 0,C 180,E1 -5460.274,E2 -5460.274} C_VEL
LIN {X 0,Y 509.93,Z 132.797,A -85,B 0,C 180,E1 -5462.419,E2 -5462.419} C_VEL
LIN {X 0,Y 512.909,Z 146.303,A -85,B 0,C 180,E1 -5464.582,E2 -5464.582} C_VEL
LIN {X 0,Y 512.19,Z 165.067,A -85,B 0,C 180,E1 -5467.25,E2 -5467.25} C_VEL
LIN {X 0,Y 512.013,Z 169.67,A -85,B 0,C 180,E1 -5467.876,E2 -5467.876} C_VEL
LIN {X 0,Y 515.325,Z 185.778,A -85,B 0,C 180,E1 -5468.289,E2 -5468.289} C_VEL
LIN {X 0,Y 514.198,Z 335.503,A -85,B 0,C 180,E1 -5470.449,E2 -5470.449} C_VEL
LIN {X 0,Y 513.801,Z 351.236,A -85,B 0,C 180,E1 -5470.835,E2 -5470.835} C_VEL
LIN {X 0,Y 513.398,Z 366.58,A -85,B 0,C 180,E1 -5471.39,E2 -5471.39} C_VEL
LIN {X 0,Y 512.859,Z 380.344,A -85,B 0,C 180,E1 -5472.041,E2 -5472.041} C_VEL
LIN {X 0,Y 512.309,Z 393.829,A -85,B 0,C 180,E1 -5472.846,E2 -5472.846} C_VEL
LIN {X 0,Y 511.752,Z 407.554,A -85,B 0,C 180,E1 -5473.853,E2 -5473.853} C_VEL
LIN {X 0,Y 511.118,Z 419.972,A -85,B 0,C 180,E1 -5474.957,E2 -5474.957} C_VEL
LIN {X 0,Y 510.608,Z 432.147,A -85,B 0,C 180,E1 -5476.265,E2 -5476.265} C_VEL
LIN {X 0,Y 510.146,Z 442.969,A -85,B 0,C 180,E1 -5477.67,E2 -5477.67} C_VEL
LIN {X 0,Y 509.873,Z 451.979,A -85,B 0,C 180,E1 -5479.075,E2 -5479.075} C_VEL
LIN {X 0,Y 509.536,Z 459.449,A -85,B 0,C 180,E1 -5480.473,E2 -5480.473} C_VEL
LIN {X 0,Y 509.376,Z 466.418,A -85,B 0,C 180,E1 -5482.069,E2 -5482.069} C_VEL
LIN {X 0,Y 509.266,Z 471.896,A -85,B 0,C 180,E1 -5483.661,E2 -5483.661} C_VEL
LIN {X 0,Y 509.159,Z 476.036,A -85,B 0,C 180,E1 -5485.249,E2 -5485.249} C_VEL
LIN {X 0,Y 509.185,Z 478.939,A -85,B 0,C 180,E1 -5486.835,E2 -5486.835} C_VEL
LIN {X 0,Y 509.11,Z 480.669,A -85,B 0,C 180,E1 -5488.418,E2 -5488.418} C_VEL
LIN {X 0,Y 509.062,Z 481.262,A -85,B 0,C 180,E1 -5490,E2 -5490} C_VEL
LIN {X 0,Y 509.11,Z 480.667,A -85,B 0,C 180,E1 -5491.582,E2 -5491.582} C_VEL
LIN {X 0,Y 509.185,Z 478.934,A -85,B 0,C 180,E1 -5493.165,E2 -5493.165} C_VEL
LIN {X 0,Y 509.159,Z 476.034,A -85,B 0,C 180,E1 -5494.751,E2 -5494.751} C_VEL
LIN {X 0,Y 509.305,Z 471.901,A -85,B 0,C 180,E1 -5496.338,E2 -5496.338} C_VEL
LIN {X 0,Y 509.376,Z 466.42,A -85,B 0,C 180,E1 -5497.931,E2 -5497.931} C_VEL
LIN {X 0,Y 509.536,Z 459.443,A -85,B 0,C 180,E1 -5499.527,E2 -5499.527} C_VEL
LIN {X 0,Y 509.881,Z 451.976,A -85,B 0,C 180,E1 -5500.925,E2 -5500.925} C_VEL
LIN {X 0,Y 510.142,Z 442.97,A -85,B 0,C 180,E1 -5502.33,E2 -5502.33} C_VEL
LIN {X 0,Y 510.608,Z 432.147,A -85,B 0,C 180,E1 -5503.735,E2 -5503.735} C_VEL
LIN {X 0,Y 511.165,Z 419.979,A -85,B 0,C 180,E1 -5505.041,E2 -5505.041} C_VEL
LIN {X 0,Y 511.739,Z 407.565,A -85,B 0,C 180,E1 -5506.147,E2 -5506.147} C_VEL
LIN {X 0,Y 512.25,Z 395.345,A -85,B 0,C 180,E1 -5507.053,E2 -5507.053} C_VEL
LIN {X 0,Y 512.762,Z 382.15,A -85,B 0,C 180,E1 -5507.859,E2 -5507.859} C_VEL
LIN {X 0,Y 513.384,Z 367.722,A -85,B 0,C 180,E1 -5508.559,E2 -5508.559} C_VEL
LIN {X 0,Y 513.758,Z 353.554,A -85,B 0,C 180,E1 -5509.088,E2 -5509.088} C_VEL
LIN {X 0,Y 514.108,Z 338.875,A -85,B 0,C 180,E1 -5509.479,E2 -5509.479} C_VEL
LIN {X 0,Y 514.345,Z 317.262,A -85,B 0,C 180,E1 -5509.831,E2 -5509.831} C_VEL
LIN {X 0,Y 515.275,Z 185.671,A -85,B 0,C 180,E1 -5511.715,E2 -5511.715} C_VEL
LIN {X 0,Y 512.042,Z 169.973,A -85,B 0,C 180,E1 -5512.103,E2 -5512.103} C_VEL
LIN {X 0,Y 512.37,Z 160.186,A -85,B 0,C 180,E1 -5513.44,E2 -5513.44} C_VEL
LIN {X 0,Y 512.926,Z 146.744,A -85,B 0,C 180,E1 -5515.352,E2 -5515.352} C_VEL
LIN {X 0,Y 510.746,Z 136.253,A -85,B 0,C 180,E1 -5517.006,E2 -5517.006} C_VEL
LIN {X 0,Y 509.929,Z 132.703,A -85,B 0,C 180,E1 -5517.609,E2 -5517.609} C_VEL
LIN {X 0,Y 509.846,Z 132.594,A -85,B 0,C 180,E1 -5520.666,E2 -5520.666} C_VEL
LIN {X 0,Y 509.859,Z 132.593,A -85,B 0,C 180,E1 -5523.461,E2 -5523.461} C_VEL
LIN {X 0,Y 509.825,Z 132.603,A -85,B 0,C 180,E1 -5526.353,E2 -5526.353} C_VEL
LIN {X 0,Y 509.848,Z 132.595,A -85,B 0,C 180,E1 -5529.352,E2 -5529.352} C_VEL
LIN {X 0,Y 509.833,Z 132.598,A -85,B 0,C 180,E1 -5532.49,E2 -5532.49} C_VEL
LIN {X 0,Y 509.839,Z 132.597,A -85,B 0,C 180,E1 -5535.33,E2 -5535.33} C_VEL
LIN {X 0,Y 509.856,Z 132.589,A -85,B 0,C 180,E1 -5538.575,E2 -5538.575} C_VEL
LIN {X 0,Y 509.852,Z 132.603,A -85,B 0,C 180,E1 -5541.787,E2 -5541.787} C_VEL
LIN {X 0,Y 509.83,Z 132.597,A -85,B 0,C 180,E1 -5544.622,E2 -5544.622} C_VEL
LIN {X 0,Y 509.861,Z 132.583,A -85,B 0,C 180,E1 -5547.481,E2 -5547.481} C_VEL
LIN {X 0,Y 509.859,Z 132.595,A -85,B 0,C 180,E1 -5550.274,E2 -5550.274} C_VEL
LIN {X 0,Y 509.884,Z 132.596,A -85,B 0,C 180,E1 -5552.944,E2 -5552.944} C_VEL
LIN {X 0,Y 509.863,Z 132.599,A -85,B 0,C 180,E1 -5555.574,E2 -5555.574} C_VEL
LIN {X 0,Y 509.852,Z 132.598,A -85,B 0,C 180,E1 -5558.998,E2 -5558.998} C_VEL
LIN {X 0,Y 509.858,Z 132.598,A -85,B 0,C 180,E1 -5561.516,E2 -5561.516} C_VEL
LIN {X 0,Y 509.913,Z 132.589,A -85,B 0,C 180,E1 -5564.819,E2 -5564.819} C_VEL
LIN {X 0,Y 509.903,Z 132.591,A -85,B 0,C 180,E1 -5568.124,E2 -5568.124} C_VEL
LIN {X 0,Y 509.905,Z 132.589,A -85,B 0,C 180,E1 -5571.28,E2 -5571.28} C_VEL
LIN {X 0,Y 509.977,Z 132.586,A -85,B 0,C 180,E1 -5574.464,E2 -5574.464} C_VEL
LIN {X 0,Y 510.052,Z 132.568,A -85,B 0,C 180,E1 -5577.631,E2 -5577.631} C_VEL
LIN {X 0,Y 510.063,Z 132.57,A -85,B 0,C 180,E1 -5580.79,E2 -5580.79} C_VEL
LIN {X 0,Y 509.917,Z 132.585,A -85,B 0,C 180,E1 -5583.16,E2 -5583.16} C_VEL
LIN {X 0,Y 509.939,Z 132.592,A -85,B 0,C 180,E1 -5586.33,E2 -5586.33} C_VEL
LIN {X 0,Y 509.911,Z 132.587,A -85,B 0,C 180,E1 -5588.72,E2 -5588.72} C_VEL
LIN {X 0,Y 509.906,Z 132.595,A -85,B 0,C 180,E1 -5591.932,E2 -5591.932} C_VEL
LIN {X 0,Y 509.897,Z 132.586,A -85,B 0,C 180,E1 -5595.242,E2 -5595.242} C_VEL
LIN {X 0,Y 509.839,Z 132.598,A -85,B 0,C 180,E1 -5598.485,E2 -5598.485} C_VEL
LIN {X 0,Y 509.848,Z 132.594,A -85,B 0,C 180,E1 -5601.002,E2 -5601.002} C_VEL
LIN {X 0,Y 509.819,Z 132.605,A -85,B 0,C 180,E1 -5603.564,E2 -5603.564} C_VEL
LIN {X 0,Y 509.82,Z 132.601,A -85,B 0,C 180,E1 -5606.357,E2 -5606.357} C_VEL
LIN {X 0,Y 509.839,Z 132.597,A -85,B 0,C 180,E1 -5608.847,E2 -5608.847} C_VEL
LIN {X 0,Y 509.818,Z 132.588,A -85,B 0,C 180,E1 -5611.59,E2 -5611.59} C_VEL
LIN {X 0,Y 509.835,Z 132.595,A -85,B 0,C 180,E1 -5614.415,E2 -5614.415} C_VEL
LIN {X 0,Y 509.808,Z 132.609,A -85,B 0,C 180,E1 -5617.342,E2 -5617.342} C_VEL
LIN {X 0,Y 509.814,Z 132.587,A -85,B 0,C 180,E1 -5620.385,E2 -5620.385} C_VEL
LIN {X 0,Y 509.806,Z 132.606,A -85,B 0,C 180,E1 -5623.573,E2 -5623.573} C_VEL
LIN {X 0,Y 509.806,Z 132.596,A -85,B 0,C 180,E1 -5626.427,E2 -5626.427} C_VEL
LIN {X 0,Y 509.814,Z 132.598,A -85,B 0,C 180,E1 -5629.615,E2 -5629.615} C_VEL
LIN {X 0,Y 509.806,Z 132.607,A -85,B 0,C 180,E1 -5632.658,E2 -5632.658} C_VEL
LIN {X 0,Y 509.8,Z 132.602,A -85,B 0,C 180,E1 -5633.721,E2 -5633.721} C_VEL
LIN {X 0,Y 509.139,Z 132.686,A -85,B 0,C 180,E1 -5634.38,E2 -5634.38} C_VEL
LIN {X 0,Y 506.339,Z 133.037,A -85,B 0,C 180,E1 -5635.453,E2 -5635.453} C_VEL
LIN {X 0,Y 503.956,Z 133.336,A -85,B 0,C 180,E1 -5636.316,E2 -5636.316} C_VEL
LIN {X 0,Y 502.906,Z 133.466,A -85,B 0,C 180,E1 -5636.983,E2 -5636.983} C_VEL
LIN {X 0,Y 502.806,Z 133.477,A -85,B 0,C 180,E1 -5637.208,E2 -5637.208} C_VEL
LIN {X 0,Y 502.744,Z 133.468,A -85,B 0,C 180,E1 -5640.079,E2 -5640.079} C_VEL
LIN {X 0,Y 502.775,Z 133.549,A -85,B 0,C 180,E1 -5643.166,E2 -5643.166} C_VEL
LIN {X 0,Y 503.042,Z 134.826,A -85,B 0,C 180,E1 -5643.444,E2 -5643.444} C_VEL
LIN {X 0,Y 505.635,Z 146.127,A -85,B 0,C 180,E1 -5645.356,E2 -5645.356} C_VEL
LIN {X 0,Y 505.596,Z 153.374,A -85,B 0,C 180,E1 -5646.469,E2 -5646.469} C_VEL
LIN {X 0,Y 505.302,Z 161.404,A -85,B 0,C 180,E1 -5647.633,E2 -5647.633} C_VEL
LIN {X 0,Y 508.732,Z 177.44,A -85,B 0,C 180,E1 -5648.047,E2 -5648.047} C_VEL
LIN {X 0,Y 507.552,Z 325.63,A -85,B 0,C 180,E1 -5650.211,E2 -5650.211} C_VEL
LIN {X 0,Y 507.188,Z 340.733,A -85,B 0,C 180,E1 -5650.576,E2 -5650.576} C_VEL
LIN {X 0,Y 506.832,Z 355.218,A -85,B 0,C 180,E1 -5651.087,E2 -5651.087} C_VEL
LIN {X 0,Y 506.263,Z 368.449,A -85,B 0,C 180,E1 -5651.695,E2 -5651.695} C_VEL
LIN {X 0,Y 505.688,Z 382.482,A -85,B 0,C 180,E1 -5652.51,E2 -5652.51} C_VEL
LIN {X 0,Y 505.085,Z 395.306,A -85,B 0,C 180,E1 -5653.426,E2 -5653.426} C_VEL
LIN {X 0,Y 504.488,Z 407.563,A -85,B 0,C 180,E1 -5654.484,E2 -5654.484} C_VEL
LIN {X 0,Y 503.914,Z 419.018,A -85,B 0,C 180,E1 -5655.667,E2 -5655.667} C_VEL
LIN {X 0,Y 503.432,Z 429,A -85,B 0,C 180,E1 -5656.888,E2 -5656.888} C_VEL
LIN {X 0,Y 503.039,Z 437.485,A -85,B 0,C 180,E1 -5658.11,E2 -5658.11} C_VEL
LIN {X 0,Y 502.751,Z 445.779,A -85,B 0,C 180,E1 -5659.53,E2 -5659.53} C_VEL
LIN {X 0,Y 502.447,Z 453.583,A -85,B 0,C 180,E1 -5661.149,E2 -5661.149} C_VEL
LIN {X 0,Y 502.246,Z 459.799,A -85,B 0,C 180,E1 -5662.765,E2 -5662.765} C_VEL
LIN {X 0,Y 502.222,Z 464.601,A -85,B 0,C 180,E1 -5664.378,E2 -5664.378} C_VEL
LIN {X 0,Y 502.099,Z 468.124,A -85,B 0,C 180,E1 -5665.987,E2 -5665.987} C_VEL
LIN {X 0,Y 502.088,Z 470.456,A -85,B 0,C 180,E1 -5667.593,E2 -5667.593} C_VEL
LIN {X 0,Y 501.987,Z 471.651,A -85,B 0,C 180,E1 -5669.198,E2 -5669.198} C_VEL
LIN {X 0,Y 501.988,Z 471.669,A -85,B 0,C 180,E1 -5670.802,E2 -5670.802} C_VEL
LIN {X 0,Y 502.089,Z 470.549,A -85,B 0,C 180,E1 -5672.407,E2 -5672.407} C_VEL
LIN {X 0,Y 502.099,Z 468.29,A -85,B 0,C 180,E1 -5674.013,E2 -5674.013} C_VEL
LIN {X 0,Y 502.213,Z 464.837,A -85,B 0,C 180,E1 -5675.622,E2 -5675.622} C_VEL
LIN {X 0,Y 502.246,Z 460.111,A -85,B 0,C 180,E1 -5677.235,E2 -5677.235} C_VEL
LIN {X 0,Y 502.443,Z 453.987,A -85,B 0,C 180,E1 -5678.851,E2 -5678.851} C_VEL
LIN {X 0,Y 502.748,Z 446.277,A -85,B 0,C 180,E1 -5680.471,E2 -5680.471} C_VEL
LIN {X 0,Y 502.998,Z 438.216,A -85,B 0,C 180,E1 -5681.868,E2 -5681.868} C_VEL
LIN {X 0,Y 503.477,Z 428.161,A -85,B 0,C 180,E1 -5683.316,E2 -5683.316} C_VEL
LIN {X 0,Y 503.973,Z 418.014,A -85,B 0,C 180,E1 -5684.538,E2 -5684.538} C_VEL
LIN {X 0,Y 504.557,Z 406.889,A -85,B 0,C 180,E1 -5685.668,E2 -5685.668} C_VEL
LIN {X 0,Y 505.092,Z 395.124,A -85,B 0,C 180,E1 -5686.677,E2 -5686.677} C_VEL
LIN {X 0,Y 505.742,Z 382.268,A -85,B 0,C 180,E1 -5687.593,E2 -5687.593} C_VEL
LIN {X 0,Y 506.302,Z 368.174,A -85,B 0,C 180,E1 -5688.409,E2 -5688.409} C_VEL
LIN {X 0,Y 506.891,Z 353.721,A -85,B 0,C 180,E1 -5689.061,E2 -5689.061} C_VEL
LIN {X 0,Y 507.242,Z 338.823,A -85,B 0,C 180,E1 -5689.567,E2 -5689.567} C_VEL
LIN {X 0,Y 507.586,Z 323.869,A -85,B 0,C 180,E1 -5689.909,E2 -5689.909} C_VEL
LIN {X 0,Y 508.734,Z 177.405,A -85,B 0,C 180,E1 -5692.044,E2 -5692.044} C_VEL
LIN {X 0,Y 505.314,Z 161.314,A -85,B 0,C 180,E1 -5692.463,E2 -5692.463} C_VEL
LIN {X 0,Y 505.829,Z 148.142,A -85,B 0,C 180,E1 -5694.415,E2 -5694.415} C_VEL
LIN {X 0,Y 504.86,Z 142.643,A -85,B 0,C 180,E1 -5695.319,E2 -5695.319} C_VEL
LIN {X 0,Y 502.783,Z 133.631,A -85,B 0,C 180,E1 -5696.896,E2 -5696.896} C_VEL
LIN {X 0,Y 502.744,Z 133.468,A -85,B 0,C 180,E1 -5699.921,E2 -5699.921} C_VEL
LIN {X 0,Y 502.799,Z 133.481,A -85,B 0,C 180,E1 -5703.034,E2 -5703.034} C_VEL
LIN {X 0,Y 502.747,Z 133.48,A -85,B 0,C 180,E1 -5705.953,E2 -5705.953} C_VEL
LIN {X 0,Y 502.78,Z 133.48,A -85,B 0,C 180,E1 -5708.978,E2 -5708.978} C_VEL
LIN {X 0,Y 502.745,Z 133.484,A -85,B 0,C 180,E1 -5712.192,E2 -5712.192} C_VEL
LIN {X 0,Y 502.786,Z 133.477,A -85,B 0,C 180,E1 -5715.47,E2 -5715.47} C_VEL
LIN {X 0,Y 502.762,Z 133.471,A -85,B 0,C 180,E1 -5718.928,E2 -5718.928} C_VEL
LIN {X 0,Y 502.772,Z 133.475,A -85,B 0,C 180,E1 -5722.044,E2 -5722.044} C_VEL
LIN {X 0,Y 502.792,Z 133.475,A -85,B 0,C 180,E1 -5725.034,E2 -5725.034} C_VEL
LIN {X 0,Y 502.783,Z 133.46,A -85,B 0,C 180,E1 -5727.915,E2 -5727.915} C_VEL
LIN {X 0,Y 502.805,Z 133.477,A -85,B 0,C 180,E1 -5730.711,E2 -5730.711} C_VEL
LIN {X 0,Y 502.776,Z 133.478,A -85,B 0,C 180,E1 -5733.46,E2 -5733.46} C_VEL
LIN {X 0,Y 502.768,Z 133.48,A -85,B 0,C 180,E1 -5736.085,E2 -5736.085} C_VEL
LIN {X 0,Y 502.78,Z 133.476,A -85,B 0,C 180,E1 -5738.689,E2 -5738.689} C_VEL
LIN {X 0,Y 502.809,Z 133.471,A -85,B 0,C 180,E1 -5741.247,E2 -5741.247} C_VEL
LIN {X 0,Y 502.837,Z 133.466,A -85,B 0,C 180,E1 -5744.665,E2 -5744.665} C_VEL
LIN {X 0,Y 502.879,Z 133.472,A -85,B 0,C 180,E1 -5748.039,E2 -5748.039} C_VEL
LIN {X 0,Y 502.864,Z 133.463,A -85,B 0,C 180,E1 -5751.156,E2 -5751.156} C_VEL
LIN {X 0,Y 502.927,Z 133.46,A -85,B 0,C 180,E1 -5754.386,E2 -5754.386} C_VEL
LIN {X 0,Y 503.019,Z 133.446,A -85,B 0,C 180,E1 -5757.598,E2 -5757.598} C_VEL
LIN {X 0,Y 502.973,Z 133.453,A -85,B 0,C 180,E1 -5760.801,E2 -5760.801} C_VEL
LIN {X 0,Y 503.021,Z 133.443,A -85,B 0,C 180,E1 -5762.402,E2 -5762.402} C_VEL
LIN {X 0,Y 502.93,Z 133.463,A -85,B 0,C 180,E1 -5765.613,E2 -5765.613} C_VEL
LIN {X 0,Y 502.866,Z 133.466,A -85,B 0,C 180,E1 -5768.843,E2 -5768.843} C_VEL
LIN {X 0,Y 502.847,Z 133.469,A -85,B 0,C 180,E1 -5772.102,E2 -5772.102} C_VEL
LIN {X 0,Y 502.851,Z 133.467,A -85,B 0,C 180,E1 -5775.4,E2 -5775.4} C_VEL
LIN {X 0,Y 502.824,Z 133.477,A -85,B 0,C 180,E1 -5778.752,E2 -5778.752} C_VEL
LIN {X 0,Y 502.785,Z 133.477,A -85,B 0,C 180,E1 -5781.311,E2 -5781.311} C_VEL
LIN {X 0,Y 502.771,Z 133.479,A -85,B 0,C 180,E1 -5783.915,E2 -5783.915} C_VEL
LIN {X 0,Y 502.838,Z 133.47,A -85,B 0,C 180,E1 -5786.567,E2 -5786.567} C_VEL
LIN {X 0,Y 502.825,Z 133.472,A -85,B 0,C 180,E1 -5789.288,E2 -5789.288} C_VEL
LIN {X 0,Y 502.783,Z 133.468,A -85,B 0,C 180,E1 -5792.085,E2 -5792.085} C_VEL
LIN {X 0,Y 502.797,Z 133.476,A -85,B 0,C 180,E1 -5794.966,E2 -5794.966} C_VEL
LIN {X 0,Y 502.794,Z 133.478,A -85,B 0,C 180,E1 -5797.954,E2 -5797.954} C_VEL
LIN {X 0,Y 502.821,Z 133.467,A -85,B 0,C 180,E1 -5801.066,E2 -5801.066} C_VEL
LIN {X 0,Y 502.787,Z 133.477,A -85,B 0,C 180,E1 -5804.53,E2 -5804.53} C_VEL
LIN {X 0,Y 502.796,Z 133.478,A -85,B 0,C 180,E1 -5807.86,E2 -5807.86} C_VEL
LIN {X 0,Y 502.803,Z 133.472,A -85,B 0,C 180,E1 -5811.024,E2 -5811.024} C_VEL
LIN {X 0,Y 502.776,Z 133.479,A -85,B 0,C 180,E1 -5814.169,E2 -5814.169} C_VEL
LIN {X 0,Y 502.833,Z 133.467,A -85,B 0,C 180,E1 -5816.993,E2 -5816.993} C_VEL
LIN {X 0,Y 502.816,Z 133.481,A -85,B 0,C 180,E1 -5820.065,E2 -5820.065} C_VEL
LIN {X 0,Y 502.887,Z 133.673,A -85,B 0,C 180,E1 -5822.141,E2 -5822.141} C_VEL
LIN {X 0,Y 505.872,Z 146.685,A -85,B 0,C 180,E1 -5824.269,E2 -5824.269} C_VEL
LIN {X 0,Y 506.069,Z 149.226,A -85,B 0,C 180,E1 -5824.654,E2 -5824.654} C_VEL
LIN {X 0,Y 505.216,Z 169.607,A -85,B 0,C 180,E1 -5827.562,E2 -5827.562} C_VEL
LIN {X 0,Y 508.639,Z 186.574,A -85,B 0,C 180,E1 -5828.002,E2 -5828.002} C_VEL
LIN {X 0,Y 507.879,Z 294.832,A -85,B 0,C 180,E1 -5829.575,E2 -5829.575} C_VEL
LIN {X 0,Y 507.473,Z 336.744,A -85,B 0,C 180,E1 -5830.208,E2 -5830.208} C_VEL
LIN {X 0,Y 507.061,Z 352.132,A -85,B 0,C 180,E1 -5830.603,E2 -5830.603} C_VEL
LIN {X 0,Y 506.635,Z 366.701,A -85,B 0,C 180,E1 -5831.14,E2 -5831.14} C_VEL
LIN {X 0,Y 506.093,Z 380.278,A -85,B 0,C 180,E1 -5831.793,E2 -5831.793} C_VEL
LIN {X 0,Y 505.517,Z 393.763,A -85,B 0,C 180,E1 -5832.608,E2 -5832.608} C_VEL
LIN {X 0,Y 504.882,Z 407.487,A -85,B 0,C 180,E1 -5833.627,E2 -5833.627} C_VEL
LIN {X 0,Y 504.227,Z 419.905,A -85,B 0,C 180,E1 -5834.747,E2 -5834.747} C_VEL
LIN {X 0,Y 503.656,Z 432.08,A -85,B 0,C 180,E1 -5836.072,E2 -5836.072} C_VEL
LIN {X 0,Y 503.157,Z 442.902,A -85,B 0,C 180,E1 -5837.496,E2 -5837.496} C_VEL
LIN {X 0,Y 502.852,Z 451.912,A -85,B 0,C 180,E1 -5838.92,E2 -5838.92} C_VEL
LIN {X 0,Y 502.472,Z 459.382,A -85,B 0,C 180,E1 -5840.338,E2 -5840.338} C_VEL
LIN {X 0,Y 502.317,Z 466.352,A -85,B 0,C 180,E1 -5841.957,E2 -5841.957} C_VEL
LIN {X 0,Y 502.17,Z 472.478,A -85,B 0,C 180,E1 -5843.784,E2 -5843.784} C_VEL
LIN {X 0,Y 502.082,Z 475.97,A -85,B 0,C 180,E1 -5845.182,E2 -5845.182} C_VEL
LIN {X 0,Y 502.102,Z 478.872,A -85,B 0,C 180,E1 -5846.79,E2 -5846.79} C_VEL
LIN {X 0,Y 502.033,Z 480.603,A -85,B 0,C 180,E1 -5848.396,E2 -5848.396} C_VEL
LIN {X 0,Y 501.977,Z 481.196,A -85,B 0,C 180,E1 -5850,E2 -5850} C_VEL
LIN {X 0,Y 502.033,Z 480.6,A -85,B 0,C 180,E1 -5851.604,E2 -5851.604} C_VEL
LIN {X 0,Y 502.102,Z 478.867,A -85,B 0,C 180,E1 -5853.21,E2 -5853.21} C_VEL
LIN {X 0,Y 502.082,Z 475.968,A -85,B 0,C 180,E1 -5854.818,E2 -5854.818} C_VEL
LIN {X 0,Y 502.233,Z 471.834,A -85,B 0,C 180,E1 -5856.428,E2 -5856.428} C_VEL
LIN {X 0,Y 502.317,Z 466.353,A -85,B 0,C 180,E1 -5858.043,E2 -5858.043} C_VEL
LIN {X 0,Y 502.472,Z 459.376,A -85,B 0,C 180,E1 -5859.662,E2 -5859.662} C_VEL
LIN {X 0,Y 502.858,Z 451.909,A -85,B 0,C 180,E1 -5861.08,E2 -5861.08} C_VEL
LIN {X 0,Y 503.155,Z 442.903,A -85,B 0,C 180,E1 -5862.504,E2 -5862.504} C_VEL
LIN {X 0,Y 503.657,Z 432.08,A -85,B 0,C 180,E1 -5863.928,E2 -5863.928} C_VEL
LIN {X 0,Y 504.217,Z 419.911,A -85,B 0,C 180,E1 -5865.253,E2 -5865.253} C_VEL
LIN {X 0,Y 504.876,Z 407.498,A -85,B 0,C 180,E1 -5866.373,E2 -5866.373} C_VEL
LIN {X 0,Y 505.44,Z 395.279,A -85,B 0,C 180,E1 -5867.29,E2 -5867.29} C_VEL
LIN {X 0,Y 505.981,Z 382.083,A -85,B 0,C 180,E1 -5868.107,E2 -5868.107} C_VEL
LIN {X 0,Y 506.643,Z 367.772,A -85,B 0,C 180,E1 -5868.81,E2 -5868.81} C_VEL
LIN {X 0,Y 507.048,Z 352.867,A -85,B 0,C 180,E1 -5869.372,E2 -5869.372} C_VEL
LIN {X 0,Y 507.437,Z 337.774,A -85,B 0,C 180,E1 -5869.77,E2 -5869.77} C_VEL
LIN {X 0,Y 507.719,Z 312.268,A -85,B 0,C 180,E1 -5870.174,E2 -5870.174} C_VEL
LIN {X 0,Y 508.651,Z 186.623,A -85,B 0,C 180,E1 -5871.997,E2 -5871.997} C_VEL
LIN {X 0,Y 505.222,Z 169.908,A -85,B 0,C 180,E1 -5872.417,E2 -5872.417} C_VEL
LIN {X 0,Y 505.567,Z 160.121,A -85,B 0,C 180,E1 -5873.774,E2 -5873.774} C_VEL
LIN {X 0,Y 506.073,Z 148.175,A -85,B 0,C 180,E1 -5875.5,E2 -5875.5} C_VEL
LIN {X 0,Y 503.126,Z 134.688,A -85,B 0,C 180,E1 -5877.675,E2 -5877.675} C_VEL
LIN {X 0,Y 502.885,Z 133.541,A -85,B 0,C 180,E1 -5877.916,E2 -5877.916} C_VEL
LIN {X 0,Y 502.796,Z 133.463,A -85,B 0,C 180,E1 -5881.143,E2 -5881.143} C_VEL
LIN {X 0,Y 502.804,Z 133.479,A -85,B 0,C 180,E1 -5883.994,E2 -5883.994} C_VEL
LIN {X 0,Y 502.778,Z 133.479,A -85,B 0,C 180,E1 -5887.178,E2 -5887.178} C_VEL
LIN {X 0,Y 502.788,Z 133.477,A -85,B 0,C 180,E1 -5890.015,E2 -5890.015} C_VEL
LIN {X 0,Y 502.803,Z 133.476,A -85,B 0,C 180,E1 -5892.199,E2 -5892.199} C_VEL
LIN {X 0,Y 502.786,Z 133.477,A -85,B 0,C 180,E1 -5895.47,E2 -5895.47} C_VEL
LIN {X 0,Y 502.82,Z 133.466,A -85,B 0,C 180,E1 -5898.934,E2 -5898.934} C_VEL
LIN {X 0,Y 502.794,Z 133.479,A -85,B 0,C 180,E1 -5902.046,E2 -5902.046} C_VEL
LIN {X 0,Y 502.796,Z 133.475,A -85,B 0,C 180,E1 -5905.034,E2 -5905.034} C_VEL
LIN {X 0,Y 502.783,Z 133.469,A -85,B 0,C 180,E1 -5907.915,E2 -5907.915} C_VEL
LIN {X 0,Y 502.824,Z 133.472,A -85,B 0,C 180,E1 -5910.712,E2 -5910.712} C_VEL
LIN {X 0,Y 502.864,Z 133.467,A -85,B 0,C 180,E1 -5913.439,E2 -5913.439} C_VEL
LIN {X 0,Y 502.785,Z 133.477,A -85,B 0,C 180,E1 -5916.086,E2 -5916.086} C_VEL
LIN {X 0,Y 502.785,Z 133.477,A -85,B 0,C 180,E1 -5918.689,E2 -5918.689} C_VEL
LIN {X 0,Y 502.824,Z 133.477,A -85,B 0,C 180,E1 -5921.248,E2 -5921.248} C_VEL
LIN {X 0,Y 502.85,Z 133.467,A -85,B 0,C 180,E1 -5924.6,E2 -5924.6} C_VEL
LIN {X 0,Y 502.878,Z 133.465,A -85,B 0,C 180,E1 -5928.039,E2 -5928.039} C_VEL
LIN {X 0,Y 502.866,Z 133.467,A -85,B 0,C 180,E1 -5931.157,E2 -5931.157} C_VEL
LIN {X 0,Y 502.93,Z 133.463,A -85,B 0,C 180,E1 -5934.387,E2 -5934.387} C_VEL
LIN {X 0,Y 503.021,Z 133.443,A -85,B 0,C 180,E1 -5937.598,E2 -5937.598} C_VEL
LIN {X 0,Y 503.012,Z 133.448,A -85,B 0,C 180,E1 -5940.801,E2 -5940.801} C_VEL
LIN {X 0,Y 503.019,Z 133.446,A -85,B 0,C 180,E1 -5942.402,E2 -5942.402} C_VEL
LIN {X 0,Y 502.927,Z 133.459,A -85,B 0,C 180,E1 -5945.614,E2 -5945.614} C_VEL
LIN {X 0,Y 502.869,Z 133.463,A -85,B 0,C 180,E1 -5948.843,E2 -5948.843} C_VEL
LIN {X 0,Y 502.847,Z 133.477,A -85,B 0,C 180,E1 -5952.102,E2 -5952.102} C_VEL
LIN {X 0,Y 502.848,Z 133.465,A -85,B 0,C 180,E1 -5955.4,E2 -5955.4} C_VEL
LIN {X 0,Y 502.812,Z 133.471,A -85,B 0,C 180,E1 -5958.753,E2 -5958.753} C_VEL
LIN {X 0,Y 502.783,Z 133.475,A -85,B 0,C 180,E1 -5961.311,E2 -5961.311} C_VEL
LIN {X 0,Y 502.768,Z 133.482,A -85,B 0,C 180,E1 -5963.915,E2 -5963.915} C_VEL
LIN {X 0,Y 502.785,Z 133.476,A -85,B 0,C 180,E1 -5966.571,E2 -5966.571} C_VEL
LIN {X 0,Y 502.811,Z 133.469,A -85,B 0,C 180,E1 -5969.934,E2 -5969.934} C_VEL
LIN {X 0,Y 502.803,Z 133.458,A -85,B 0,C 180,E1 -5973.034,E2 -5973.034} C_VEL
LIN {X 0,Y 502.767,Z 133.482,A -85,B 0,C 180,E1 -5975.952,E2 -5975.952} C_VEL
LIN {X 0,Y 502.793,Z 133.474,A -85,B 0,C 180,E1 -5978.977,E2 -5978.977} C_VEL
LIN {X 0,Y 502.745,Z 133.48,A -85,B 0,C 180,E1 -5982.192,E2 -5982.192} C_VEL
LIN {X 0,Y 502.786,Z 133.473,A -85,B 0,C 180,E1 -5985.47,E2 -5985.47} C_VEL
LIN {X 0,Y 502.765,Z 133.486,A -85,B 0,C 180,E1 -5988.928,E2 -5988.928} C_VEL
LIN {X 0,Y 502.79,Z 133.478,A -85,B 0,C 180,E1 -5992.046,E2 -5992.046} C_VEL
LIN {X 0,Y 502.788,Z 133.484,A -85,B 0,C 180,E1 -5995.033,E2 -5995.033} C_VEL
LIN {X 0,Y 502.806,Z 133.477,A -85,B 0,C 180,E1 -5997.208,E2 -5997.208} C_VEL
LIN {X 0,Y 502.092,Z 133.567,A -85,B 0,C 180,E1 -5997.877,E2 -5997.877} C_VEL
LIN {X 0,Y 499.201,Z 133.915,A -85,B 0,C 180,E1 -5998.962,E2 -5998.962} C_VEL
LIN {X 0,Y 496.787,Z 134.211,A -85,B 0,C 180,E1 -5999.836,E2 -5999.836} C_VEL
LIN {X 0,Y 495.759,Z 134.341,A -85,B 0,C 180,E1 -6000.512,E2 -6000.512} C_VEL
LIN {X 0,Y 495.679,Z 134.354,A -85,B 0,C 180,E1 -6000.74,E2 -6000.74} C_VEL
LIN {X 0,Y 495.77,Z 134.477,A -85,B 0,C 180,E1 -6002.909,E2 -6002.909} C_VEL
LIN {X 0,Y 498.469,Z 146.195,A -85,B 0,C 180,E1 -6004.977,E2 -6004.977} C_VEL
LIN {X 0,Y 498.961,Z 150.446,A -85,B 0,C 180,E1 -6005.67,E2 -6005.67} C_VEL
LIN {X 0,Y 498.464,Z 161.181,A -85,B 0,C 180,E1 -6007.285,E2 -6007.285} C_VEL
LIN {X 0,Y 499.861,Z 167.797,A -85,B 0,C 180,E1 -6007.487,E2 -6007.487} C_VEL
LIN {X 0,Y 502.213,Z 179.12,A -85,B 0,C 180,E1 -6007.77,E2 -6007.77} C_VEL
LIN {X 0,Y 500.875,Z 326.978,A -85,B 0,C 180,E1 -6009.96,E2 -6009.96} C_VEL
LIN {X 0,Y 500.475,Z 342.654,A -85,B 0,C 180,E1 -6010.361,E2 -6010.361} C_VEL
LIN {X 0,Y 500.096,Z 356.636,A -85,B 0,C 180,E1 -6010.877,E2 -6010.877} C_VEL
LIN {X 0,Y 499.452,Z 370.508,A -85,B 0,C 180,E1 -6011.542,E2 -6011.542} C_VEL
LIN {X 0,Y 498.841,Z 384.136,A -85,B 0,C 180,E1 -6012.368,E2 -6012.368} C_VEL
LIN {X 0,Y 498.193,Z 396.669,A -85,B 0,C 180,E1 -6013.296,E2 -6013.296} C_VEL
LIN {X 0,Y 497.51,Z 409.36,A -85,B 0,C 180,E1 -6014.431,E2 -6014.431} C_VEL
LIN {X 0,Y 496.919,Z 420.867,A -85,B 0,C 180,E1 -6015.67,E2 -6015.67} C_VEL
LIN {X 0,Y 496.376,Z 430.553,A -85,B 0,C 180,E1 -6016.907,E2 -6016.907} C_VEL
LIN {X 0,Y 495.976,Z 439.67,A -85,B 0,C 180,E1 -6018.287,E2 -6018.287} C_VEL
LIN {X 0,Y 495.609,Z 447.954,A -85,B 0,C 180,E1 -6019.79,E2 -6019.79} C_VEL
LIN {X 0,Y 495.34,Z 455.337,A -85,B 0,C 180,E1 -6021.432,E2 -6021.432} C_VEL
LIN {X 0,Y 495.148,Z 461.199,A -85,B 0,C 180,E1 -6023.071,E2 -6023.071} C_VEL
LIN {X 0,Y 495.138,Z 464.669,A -85,B 0,C 180,E1 -6024.298,E2 -6024.298} C_VEL
LIN {X 0,Y 494.998,Z 468.191,A -85,B 0,C 180,E1 -6025.929,E2 -6025.929} C_VEL
LIN {X 0,Y 494.995,Z 470.523,A -85,B 0,C 180,E1 -6027.559,E2 -6027.559} C_VEL
LIN {X 0,Y 494.907,Z 471.717,A -85,B 0,C 180,E1 -6029.186,E2 -6029.186} C_VEL
LIN {X 0,Y 494.908,Z 471.736,A -85,B 0,C 180,E1 -6030.814,E2 -6030.814} C_VEL
LIN {X 0,Y 494.995,Z 470.615,A -85,B 0,C 180,E1 -6032.441,E2 -6032.441} C_VEL
LIN {X 0,Y 494.998,Z 468.356,A -85,B 0,C 180,E1 -6034.071,E2 -6034.071} C_VEL
LIN {X 0,Y 495.122,Z 464.902,A -85,B 0,C 180,E1 -6035.702,E2 -6035.702} C_VEL
LIN {X 0,Y 495.171,Z 460.175,A -85,B 0,C 180,E1 -6037.339,E2 -6037.339} C_VEL
LIN {X 0,Y 495.388,Z 454.051,A -85,B 0,C 180,E1 -6038.978,E2 -6038.978} C_VEL
LIN {X 0,Y 495.744,Z 446.34,A -85,B 0,C 180,E1 -6040.62,E2 -6040.62} C_VEL
LIN {X 0,Y 496.071,Z 437.463,A -85,B 0,C 180,E1 -6042.164,E2 -6042.164} C_VEL
LIN {X 0,Y 496.524,Z 428.223,A -85,B 0,C 180,E1 -6043.506,E2 -6043.506} C_VEL
LIN {X 0,Y 497.066,Z 418.075,A -85,B 0,C 180,E1 -6044.744,E2 -6044.744} C_VEL
LIN {X 0,Y 497.67,Z 407.269,A -85,B 0,C 180,E1 -6045.859,E2 -6045.859} C_VEL
LIN {X 0,Y 498.267,Z 395.184,A -85,B 0,C 180,E1 -6046.913,E2 -6046.913} C_VEL
LIN {X 0,Y 498.959,Z 382.327,A -85,B 0,C 180,E1 -6047.84,E2 -6047.84} C_VEL
LIN {X 0,Y 499.548,Z 368.231,A -85,B 0,C 180,E1 -6048.667,E2 -6048.667} C_VEL
LIN {X 0,Y 500.208,Z 353.033,A -85,B 0,C 180,E1 -6049.356,E2 -6049.356} C_VEL
LIN {X 0,Y 500.604,Z 338.237,A -85,B 0,C 180,E1 -6049.856,E2 -6049.856} C_VEL
LIN {X 0,Y 500.917,Z 323.908,A -85,B 0,C 180,E1 -6050.185,E2 -6050.185} C_VEL
LIN {X 0,Y 502.179,Z 178.735,A -85,B 0,C 180,E1 -6052.328,E2 -6052.328} C_VEL
LIN {X 0,Y 498.487,Z 161.421,A -85,B 0,C 180,E1 -6052.786,E2 -6052.786} C_VEL
LIN {X 0,Y 498.983,Z 149.62,A -85,B 0,C 180,E1 -6054.551,E2 -6054.551} C_VEL
LIN {X 0,Y 496.958,Z 139.856,A -85,B 0,C 180,E1 -6056.204,E2 -6056.204} C_VEL
LIN {X 0,Y 495.821,Z 134.809,A -85,B 0,C 180,E1 -6057.088,E2 -6057.088} C_VEL
LIN {X 0,Y 495.74,Z 134.345,A -85,B 0,C 180,E1 -6057.321,E2 -6057.321} C_VEL
LIN {X 0,Y 495.709,Z 134.344,A -85,B 0,C 180,E1 -6060.69,E2 -6060.69} C_VEL
LIN {X 0,Y 495.739,Z 134.356,A -85,B 0,C 180,E1 -6063.566,E2 -6063.566} C_VEL
LIN {X 0,Y 495.692,Z 134.359,A -85,B 0,C 180,E1 -6066.547,E2 -6066.547} C_VEL
LIN {X 0,Y 495.74,Z 134.349,A -85,B 0,C 180,E1 -6069.64,E2 -6069.64} C_VEL
LIN {X 0,Y 495.695,Z 134.362,A -85,B 0,C 180,E1 -6072.887,E2 -6072.887} C_VEL
LIN {X 0,Y 495.723,Z 134.357,A -85,B 0,C 180,E1 -6075.998,E2 -6075.998} C_VEL
LIN {X 0,Y 495.726,Z 134.343,A -85,B 0,C 180,E1 -6079.296,E2 -6079.296} C_VEL
LIN {X 0,Y 495.728,Z 134.351,A -85,B 0,C 180,E1 -6081.406,E2 -6081.406} C_VEL
LIN {X 0,Y 495.744,Z 134.361,A -85,B 0,C 180,E1 -6084.462,E2 -6084.462} C_VEL
LIN {X 0,Y 495.753,Z 134.334,A -85,B 0,C 180,E1 -6087.404,E2 -6087.404} C_VEL
LIN {X 0,Y 495.758,Z 134.348,A -85,B 0,C 180,E1 -6090.253,E2 -6090.253} C_VEL
LIN {X 0,Y 495.741,Z 134.354,A -85,B 0,C 180,E1 -6093.27,E2 -6093.27} C_VEL
LIN {X 0,Y 495.74,Z 134.358,A -85,B 0,C 180,E1 -6096.612,E2 -6096.612} C_VEL
LIN {X 0,Y 495.781,Z 134.346,A -85,B 0,C 180,E1 -6099.324,E2 -6099.324} C_VEL
LIN {X 0,Y 495.781,Z 134.351,A -85,B 0,C 180,E1 -6101.828,E2 -6101.828} C_VEL
LIN {X 0,Y 495.782,Z 134.345,A -85,B 0,C 180,E1 -6105.217,E2 -6105.217} C_VEL
LIN {X 0,Y 495.853,Z 134.341,A -85,B 0,C 180,E1 -6108.555,E2 -6108.555} C_VEL
LIN {X 0,Y 495.832,Z 134.342,A -85,B 0,C 180,E1 -6111.851,E2 -6111.851} C_VEL
LIN {X 0,Y 495.882,Z 134.338,A -85,B 0,C 180,E1 -6114.306,E2 -6114.306} C_VEL
LIN {X 0,Y 495.986,Z 134.322,A -85,B 0,C 180,E1 -6117.564,E2 -6117.564} C_VEL
LIN {X 0,Y 496,Z 134.324,A -85,B 0,C 180,E1 -6120,E2 -6120} C_VEL
LIN {X 0,Y 495.988,Z 134.319,A -85,B 0,C 180,E1 -6122.436,E2 -6122.436} C_VEL
LIN {X 0,Y 495.885,Z 134.34,A -85,B 0,C 180,E1 -6125.694,E2 -6125.694} C_VEL
LIN {X 0,Y 495.836,Z 134.343,A -85,B 0,C 180,E1 -6128.97,E2 -6128.97} C_VEL
LIN {X 0,Y 495.831,Z 134.343,A -85,B 0,C 180,E1 -6132.035,E2 -6132.035} C_VEL
LIN {X 0,Y 495.826,Z 134.342,A -85,B 0,C 180,E1 -6135.451,E2 -6135.451} C_VEL
LIN {X 0,Y 495.78,Z 134.355,A -85,B 0,C 180,E1 -6139.028,E2 -6139.028} C_VEL
LIN {X 0,Y 495.744,Z 134.352,A -85,B 0,C 180,E1 -6141.629,E2 -6141.629} C_VEL
LIN {X 0,Y 495.718,Z 134.359,A -85,B 0,C 180,E1 -6144.277,E2 -6144.277} C_VEL
LIN {X 0,Y 495.786,Z 134.353,A -85,B 0,C 180,E1 -6146.976,E2 -6146.976} C_VEL
LIN {X 0,Y 495.767,Z 134.35,A -85,B 0,C 180,E1 -6149.746,E2 -6149.746} C_VEL
LIN {X 0,Y 495.753,Z 134.337,A -85,B 0,C 180,E1 -6152.595,E2 -6152.595} C_VEL
LIN {X 0,Y 495.748,Z 134.351,A -85,B 0,C 180,E1 -6155.538,E2 -6155.538} C_VEL
LIN {X 0,Y 495.764,Z 134.348,A -85,B 0,C 180,E1 -6158.768,E2 -6158.768} C_VEL
LIN {X 0,Y 495.757,Z 134.347,A -85,B 0,C 180,E1 -6161.781,E2 -6161.781} C_VEL
LIN {X 0,Y 495.738,Z 134.35,A -85,B 0,C 180,E1 -6165.141,E2 -6165.141} C_VEL
LIN {X 0,Y 495.757,Z 134.36,A -85,B 0,C 180,E1 -6168.219,E2 -6168.219} C_VEL
LIN {X 0,Y 495.752,Z 134.352,A -85,B 0,C 180,E1 -6171.408,E2 -6171.408} C_VEL
LIN {X 0,Y 495.749,Z 134.355,A -85,B 0,C 180,E1 -6174.462,E2 -6174.462} C_VEL
LIN {X 0,Y 495.768,Z 134.338,A -85,B 0,C 180,E1 -6177.406,E2 -6177.406} C_VEL
LIN {X 0,Y 495.767,Z 134.357,A -85,B 0,C 180,E1 -6180.254,E2 -6180.254} C_VEL
LIN {X 0,Y 495.853,Z 134.535,A -85,B 0,C 180,E1 -6181.85,E2 -6181.85} C_VEL
LIN {X 0,Y 499.184,Z 149.281,A -85,B 0,C 180,E1 -6184.297,E2 -6184.297} C_VEL
LIN {X 0,Y 498.549,Z 166.031,A -85,B 0,C 180,E1 -6186.752,E2 -6186.752} C_VEL
LIN {X 0,Y 498.419,Z 169.723,A -85,B 0,C 180,E1 -6187.252,E2 -6187.252} C_VEL
LIN {X 0,Y 502.147,Z 188.204,A -85,B 0,C 180,E1 -6187.728,E2 -6187.728} C_VEL
LIN {X 0,Y 500.855,Z 335.383,A -85,B 0,C 180,E1 -6189.906,E2 -6189.906} C_VEL
LIN {X 0,Y 500.418,Z 351.111,A -85,B 0,C 180,E1 -6190.302,E2 -6190.302} C_VEL
LIN {X 0,Y 499.941,Z 365.818,A -85,B 0,C 180,E1 -6190.841,E2 -6190.841} C_VEL
LIN {X 0,Y 499.326,Z 380.214,A -85,B 0,C 180,E1 -6191.537,E2 -6191.537} C_VEL
LIN {X 0,Y 498.71,Z 393.698,A -85,B 0,C 180,E1 -6192.363,E2 -6192.363} C_VEL
LIN {X 0,Y 497.99,Z 407.421,A -85,B 0,C 180,E1 -6193.394,E2 -6193.394} C_VEL
LIN {X 0,Y 497.342,Z 419.839,A -85,B 0,C 180,E1 -6194.53,E2 -6194.53} C_VEL
LIN {X 0,Y 496.712,Z 432.014,A -85,B 0,C 180,E1 -6195.873,E2 -6195.873} C_VEL
LIN {X 0,Y 496.167,Z 442.835,A -85,B 0,C 180,E1 -6197.317,E2 -6197.317} C_VEL
LIN {X 0,Y 495.819,Z 451.845,A -85,B 0,C 180,E1 -6198.761,E2 -6198.761} C_VEL
LIN {X 0,Y 495.418,Z 459.315,A -85,B 0,C 180,E1 -6200.199,E2 -6200.199} C_VEL
LIN {X 0,Y 495.246,Z 466.285,A -85,B 0,C 180,E1 -6201.842,E2 -6201.842} C_VEL
LIN {X 0,Y 495.088,Z 471.993,A -85,B 0,C 180,E1 -6203.555,E2 -6203.555} C_VEL
LIN {X 0,Y 495.006,Z 475.903,A -85,B 0,C 180,E1 -6205.113,E2 -6205.113} C_VEL
LIN {X 0,Y 495.021,Z 478.806,A -85,B 0,C 180,E1 -6206.744,E2 -6206.744} C_VEL
LIN {X 0,Y 494.958,Z 480.537,A -85,B 0,C 180,E1 -6208.373,E2 -6208.373} C_VEL
LIN {X 0,Y 494.895,Z 481.13,A -85,B 0,C 180,E1 -6210,E2 -6210} C_VEL
LIN {X 0,Y 494.958,Z 480.534,A -85,B 0,C 180,E1 -6211.627,E2 -6211.627} C_VEL
LIN {X 0,Y 495.021,Z 478.801,A -85,B 0,C 180,E1 -6213.256,E2 -6213.256} C_VEL
LIN {X 0,Y 495.006,Z 475.901,A -85,B 0,C 180,E1 -6214.887,E2 -6214.887} C_VEL
LIN {X 0,Y 495.162,Z 471.768,A -85,B 0,C 180,E1 -6216.52,E2 -6216.52} C_VEL
LIN {X 0,Y 495.246,Z 466.286,A -85,B 0,C 180,E1 -6218.158,E2 -6218.158} C_VEL
LIN {X 0,Y 495.418,Z 459.309,A -85,B 0,C 180,E1 -6219.801,E2 -6219.801} C_VEL
LIN {X 0,Y 495.819,Z 451.842,A -85,B 0,C 180,E1 -6221.239,E2 -6221.239} C_VEL
LIN {X 0,Y 496.166,Z 442.836,A -85,B 0,C 180,E1 -6222.683,E2 -6222.683} C_VEL
LIN {X 0,Y 496.715,Z 432.013,A -85,B 0,C 180,E1 -6224.127,E2 -6224.127} C_VEL
LIN {X 0,Y 497.325,Z 419.844,A -85,B 0,C 180,E1 -6225.47,E2 -6225.47} C_VEL
LIN {X 0,Y 498.035,Z 407.43,A -85,B 0,C 180,E1 -6226.604,E2 -6226.604} C_VEL
LIN {X 0,Y 498.615,Z 395.21,A -85,B 0,C 180,E1 -6227.535,E2 -6227.535} C_VEL
LIN {X 0,Y 499.228,Z 382.014,A -85,B 0,C 180,E1 -6228.36,E2 -6228.36} C_VEL
LIN {X 0,Y 499.888,Z 367.893,A -85,B 0,C 180,E1 -6229.065,E2 -6229.065} C_VEL
LIN {X 0,Y 500.322,Z 353.285,A -85,B 0,C 180,E1 -6229.626,E2 -6229.626} C_VEL
LIN {X 0,Y 500.73,Z 338.729,A -85,B 0,C 180,E1 -6230.022,E2 -6230.022} C_VEL
LIN {X 0,Y 501.005,Z 317.11,A -85,B 0,C 180,E1 -6230.382,E2 -6230.382} C_VEL
LIN {X 0,Y 502.064,Z 187.592,A -85,B 0,C 180,E1 -6232.285,E2 -6232.285} C_VEL
LIN {X 0,Y 498.414,Z 169.834,A -85,B 0,C 180,E1 -6232.74,E2 -6232.74} C_VEL
LIN {X 0,Y 498.781,Z 160.055,A -85,B 0,C 180,E1 -6234.118,E2 -6234.118} C_VEL
LIN {X 0,Y 499.173,Z 149.298,A -85,B 0,C 180,E1 -6235.701,E2 -6235.701} C_VEL
LIN {X 0,Y 495.916,Z 134.909,A -85,B 0,C 180,E1 -6238.074,E2 -6238.074} C_VEL
LIN {X 0,Y 495.828,Z 134.363,A -85,B 0,C 180,E1 -6238.27,E2 -6238.27} C_VEL
LIN {X 0,Y 495.755,Z 134.334,A -85,B 0,C 180,E1 -6241.636,E2 -6241.636} C_VEL
LIN {X 0,Y 495.778,Z 134.354,A -85,B 0,C 180,E1 -6244.543,E2 -6244.543} C_VEL
LIN {X 0,Y 495.73,Z 134.36,A -85,B 0,C 180,E1 -6247.562,E2 -6247.562} C_VEL
LIN {X 0,Y 495.767,Z 134.352,A -85,B 0,C 180,E1 -6250.7,E2 -6250.7} C_VEL
LIN {X 0,Y 495.728,Z 134.352,A -85,B 0,C 180,E1 -6254.002,E2 -6254.002} C_VEL
LIN {X 0,Y 495.726,Z 134.359,A -85,B 0,C 180,E1 -6257.117,E2 -6257.117} C_VEL
LIN {X 0,Y 495.759,Z 134.345,A -85,B 0,C 180,E1 -6259.953,E2 -6259.953} C_VEL
LIN {X 0,Y 495.728,Z 134.356,A -85,B 0,C 180,E1 -6262.553,E2 -6262.553} C_VEL
LIN {X 0,Y 495.771,Z 134.342,A -85,B 0,C 180,E1 -6265.456,E2 -6265.456} C_VEL
LIN {X 0,Y 495.755,Z 134.342,A -85,B 0,C 180,E1 -6268.364,E2 -6268.364} C_VEL
LIN {X 0,Y 495.788,Z 134.354,A -85,B 0,C 180,E1 -6271.507,E2 -6271.507} C_VEL
LIN {X 0,Y 495.791,Z 134.344,A -85,B 0,C 180,E1 -6273.932,E2 -6273.932} C_VEL
LIN {X 0,Y 495.761,Z 134.357,A -85,B 0,C 180,E1 -6277.14,E2 -6277.14} C_VEL
LIN {X 0,Y 495.769,Z 134.348,A -85,B 0,C 180,E1 -6280.11,E2 -6280.11} C_VEL
LIN {X 0,Y 495.758,Z 134.356,A -85,B 0,C 180,E1 -6282.68,E2 -6282.68} C_VEL
LIN {X 0,Y 495.789,Z 134.351,A -85,B 0,C 180,E1 -6285.217,E2 -6285.217} C_VEL
LIN {X 0,Y 495.853,Z 134.345,A -85,B 0,C 180,E1 -6288.555,E2 -6288.555} C_VEL
LIN {X 0,Y 495.838,Z 134.339,A -85,B 0,C 180,E1 -6291.852,E2 -6291.852} C_VEL
LIN {X 0,Y 495.885,Z 134.339,A -85,B 0,C 180,E1 -6294.307,E2 -6294.307} C_VEL
LIN {X 0,Y 495.989,Z 134.319,A -85,B 0,C 180,E1 -6297.564,E2 -6297.564} C_VEL
LIN {X 0,Y 495.963,Z 134.325,A -85,B 0,C 180,E1 -6300.812,E2 -6300.812} C_VEL
LIN {X 0,Y 495.987,Z 134.322,A -85,B 0,C 180,E1 -6302.436,E2 -6302.436} C_VEL
LIN {X 0,Y 495.883,Z 134.338,A -85,B 0,C 180,E1 -6305.694,E2 -6305.694} C_VEL
LIN {X 0,Y 495.838,Z 134.338,A -85,B 0,C 180,E1 -6308.97,E2 -6308.97} C_VEL
LIN {X 0,Y 495.831,Z 134.35,A -85,B 0,C 180,E1 -6312.035,E2 -6312.035} C_VEL
LIN {X 0,Y 495.804,Z 134.342,A -85,B 0,C 180,E1 -6315.442,E2 -6315.442} C_VEL
LIN {X 0,Y 495.773,Z 134.347,A -85,B 0,C 180,E1 -6319.029,E2 -6319.029} C_VEL
LIN {X 0,Y 495.743,Z 134.355,A -85,B 0,C 180,E1 -6321.629,E2 -6321.629} C_VEL
LIN {X 0,Y 495.714,Z 134.355,A -85,B 0,C 180,E1 -6324.277,E2 -6324.277} C_VEL
LIN {X 0,Y 495.733,Z 134.355,A -85,B 0,C 180,E1 -6326.979,E2 -6326.979} C_VEL
LIN {X 0,Y 495.76,Z 134.344,A -85,B 0,C 180,E1 -6330.146,E2 -6330.146} C_VEL
LIN {X 0,Y 495.752,Z 134.337,A -85,B 0,C 180,E1 -6333.237,E2 -6333.237} C_VEL
LIN {X 0,Y 495.712,Z 134.36,A -85,B 0,C 180,E1 -6336.087,E2 -6336.087} C_VEL
LIN {X 0,Y 495.758,Z 134.349,A -85,B 0,C 180,E1 -6338.767,E2 -6338.767} C_VEL
LIN {X 0,Y 495.724,Z 134.357,A -85,B 0,C 180,E1 -6341.785,E2 -6341.785} C_VEL
LIN {X 0,Y 495.738,Z 134.355,A -85,B 0,C 180,E1 -6345.141,E2 -6345.141} C_VEL
LIN {X 0,Y 495.724,Z 134.358,A -85,B 0,C 180,E1 -6348.215,E2 -6348.215} C_VEL
LIN {X 0,Y 495.746,Z 134.359,A -85,B 0,C 180,E1 -6351.408,E2 -6351.408} C_VEL
LIN {X 0,Y 495.739,Z 134.355,A -85,B 0,C 180,E1 -6354.462,E2 -6354.462} C_VEL
LIN {X 0,Y 495.763,Z 134.357,A -85,B 0,C 180,E1 -6357.405,E2 -6357.405} C_VEL
LIN {X 0,Y 495.695,Z 134.346,A -85,B 0,C 180,E1 -6360.249,E2 -6360.249} C_VEL
LIN {X 0,Y 495.679,Z 134.354,A -85,B 0,C 180,E1 -6360.74,E2 -6360.74} C_VEL
LIN {X 0,Y 494.988,Z 134.458,A -85,B 0,C 180,E1 -6361.211,E2 -6361.211} C_VEL
LIN {X 0,Y 492.125,Z 134.808,A -85,B 0,C 180,E1 -6361.951,E2 -6361.951} C_VEL
LIN {X 0,Y 489.93,Z 135.621,A -85,B 0,C 180,E1 -6362.519,E2 -6362.519} C_VEL
LIN {X 0,Y 489.179,Z 136.975,A -85,B 0,C 180,E1 -6362.939,E2 -6362.939} C_VEL
LIN {X 0,Y 489.239,Z 137.632,A -85,B 0,C 180,E1 -6363.071,E2 -6363.071} C_VEL
LIN {X 0,Y 492.088,Z 150.512,A -85,B 0,C 180,E1 -6365.307,E2 -6365.307} C_VEL
LIN {X 0,Y 491.664,Z 161.251,A -85,B 0,C 180,E1 -6366.953,E2 -6366.953} C_VEL
LIN {X 0,Y 493.182,Z 168.55,A -85,B 0,C 180,E1 -6367.175,E2 -6367.175} C_VEL
LIN {X 0,Y 495.621,Z 179.852,A -85,B 0,C 180,E1 -6367.468,E2 -6367.468} C_VEL
LIN {X 0,Y 494.226,Z 327.066,A -85,B 0,C 180,E1 -6369.679,E2 -6369.679} C_VEL
LIN {X 0,Y 493.778,Z 342.627,A -85,B 0,C 180,E1 -6370.08,E2 -6370.08} C_VEL
LIN {X 0,Y 493.389,Z 356.961,A -85,B 0,C 180,E1 -6370.618,E2 -6370.618} C_VEL
LIN {X 0,Y 492.7,Z 370.583,A -85,B 0,C 180,E1 -6371.28,E2 -6371.28} C_VEL
LIN {X 0,Y 492.048,Z 384.21,A -85,B 0,C 180,E1 -6372.116,E2 -6372.116} C_VEL
LIN {X 0,Y 491.359,Z 396.741,A -85,B 0,C 180,E1 -6373.057,E2 -6373.057} C_VEL
LIN {X 0,Y 490.646,Z 409.432,A -85,B 0,C 180,E1 -6374.207,E2 -6374.207} C_VEL
LIN {X 0,Y 489.985,Z 420.939,A -85,B 0,C 180,E1 -6375.463,E2 -6375.463} C_VEL
LIN {X 0,Y 489.413,Z 430.624,A -85,B 0,C 180,E1 -6376.717,E2 -6376.717} C_VEL
LIN {X 0,Y 488.945,Z 439.972,A -85,B 0,C 180,E1 -6378.156,E2 -6378.156} C_VEL
LIN {X 0,Y 488.564,Z 448.024,A -85,B 0,C 180,E1 -6379.641,E2 -6379.641} C_VEL
LIN {X 0,Y 488.284,Z 455.407,A -85,B 0,C 180,E1 -6381.308,E2 -6381.308} C_VEL
LIN {X 0,Y 488.067,Z 461.268,A -85,B 0,C 180,E1 -6382.97,E2 -6382.97} C_VEL
LIN {X 0,Y 488.054,Z 464.738,A -85,B 0,C 180,E1 -6384.215,E2 -6384.215} C_VEL
LIN {X 0,Y 487.899,Z 468.259,A -85,B 0,C 180,E1 -6385.87,E2 -6385.87} C_VEL
LIN {X 0,Y 487.905,Z 470.59,A -85,B 0,C 180,E1 -6387.523,E2 -6387.523} C_VEL
LIN {X 0,Y 487.831,Z 471.783,A -85,B 0,C 180,E1 -6389.175,E2 -6389.175} C_VEL
LIN {X 0,Y 487.831,Z 471.802,A -85,B 0,C 180,E1 -6390.826,E2 -6390.826} C_VEL
LIN {X 0,Y 487.905,Z 470.68,A -85,B 0,C 180,E1 -6392.477,E2 -6392.477} C_VEL
LIN {X 0,Y 487.898,Z 468.421,A -85,B 0,C 180,E1 -6394.13,E2 -6394.13} C_VEL
LIN {X 0,Y 488.033,Z 464.967,A -85,B 0,C 180,E1 -6395.786,E2 -6395.786} C_VEL
LIN {X 0,Y 488.119,Z 460.24,A -85,B 0,C 180,E1 -6397.446,E2 -6397.446} C_VEL
LIN {X 0,Y 488.32,Z 454.115,A -85,B 0,C 180,E1 -6399.109,E2 -6399.109} C_VEL
LIN {X 0,Y 488.74,Z 446.403,A -85,B 0,C 180,E1 -6400.774,E2 -6400.774} C_VEL
LIN {X 0,Y 489.04,Z 438.11,A -85,B 0,C 180,E1 -6402.25,E2 -6402.25} C_VEL
LIN {X 0,Y 489.592,Z 428.285,A -85,B 0,C 180,E1 -6403.701,E2 -6403.701} C_VEL
LIN {X 0,Y 490.163,Z 418.138,A -85,B 0,C 180,E1 -6404.957,E2 -6404.957} C_VEL
LIN {X 0,Y 490.847,Z 406.592,A -85,B 0,C 180,E1 -6406.16,E2 -6406.16} C_VEL
LIN {X 0,Y 491.507,Z 393.956,A -85,B 0,C 180,E1 -6407.26,E2 -6407.26} C_VEL
LIN {X 0,Y 492.229,Z 380.807,A -85,B 0,C 180,E1 -6408.2,E2 -6408.2} C_VEL
LIN {X 0,Y 492.821,Z 368.288,A -85,B 0,C 180,E1 -6408.931,E2 -6408.931} C_VEL
LIN {X 0,Y 493.495,Z 353.696,A -85,B 0,C 180,E1 -6409.605,E2 -6409.605} C_VEL
LIN {X 0,Y 493.888,Z 339.646,A -85,B 0,C 180,E1 -6410.097,E2 -6410.097} C_VEL
LIN {X 0,Y 494.21,Z 325.883,A -85,B 0,C 180,E1 -6410.436,E2 -6410.436} C_VEL
LIN {X 0,Y 495.625,Z 179.766,A -85,B 0,C 180,E1 -6412.624,E2 -6412.624} C_VEL
LIN {X 0,Y 491.701,Z 161.352,A -85,B 0,C 180,E1 -6413.127,E2 -6413.127} C_VEL
LIN {X 0,Y 492.146,Z 151.098,A -85,B 0,C 180,E1 -6414.69,E2 -6414.69} C_VEL
LIN {X 0,Y 489.411,Z 138.567,A -85,B 0,C 180,E1 -6416.859,E2 -6416.859} C_VEL
LIN {X 0,Y 488.726,Z 135.336,A -85,B 0,C 180,E1 -6417.485,E2 -6417.485} C_VEL
LIN {X 0,Y 488.651,Z 135.221,A -85,B 0,C 180,E1 -6420.351,E2 -6420.351} C_VEL
LIN {X 0,Y 488.708,Z 135.232,A -85,B 0,C 180,E1 -6423.479,E2 -6423.479} C_VEL
LIN {X 0,Y 488.652,Z 135.236,A -85,B 0,C 180,E1 -6426.349,E2 -6426.349} C_VEL
LIN {X 0,Y 488.686,Z 135.231,A -85,B 0,C 180,E1 -6429.256,E2 -6429.256} C_VEL
LIN {X 0,Y 488.667,Z 135.238,A -85,B 0,C 180,E1 -6431.594,E2 -6431.594} C_VEL
LIN {X 0,Y 488.702,Z 135.228,A -85,B 0,C 180,E1 -6434.803,E2 -6434.803} C_VEL
LIN {X 0,Y 488.651,Z 135.237,A -85,B 0,C 180,E1 -6437.47,E2 -6437.47} C_VEL
LIN {X 0,Y 488.705,Z 135.215,A -85,B 0,C 180,E1 -6439.674,E2 -6439.674} C_VEL
LIN {X 0,Y 488.667,Z 135.242,A -85,B 0,C 180,E1 -6442.84,E2 -6442.84} C_VEL
LIN {X 0,Y 488.719,Z 135.226,A -85,B 0,C 180,E1 -6445.886,E2 -6445.886} C_VEL
LIN {X 0,Y 488.69,Z 135.22,A -85,B 0,C 180,E1 -6448.82,E2 -6448.82} C_VEL
LIN {X 0,Y 488.696,Z 135.232,A -85,B 0,C 180,E1 -6451.668,E2 -6451.668} C_VEL
LIN {X 0,Y 488.7,Z 135.227,A -85,B 0,C 180,E1 -6454.959,E2 -6454.959} C_VEL
LIN {X 0,Y 488.698,Z 135.238,A -85,B 0,C 180,E1 -6458.043,E2 -6458.043} C_VEL
LIN {X 0,Y 488.732,Z 135.226,A -85,B 0,C 180,E1 -6460.686,E2 -6460.686} C_VEL
LIN {X 0,Y 488.711,Z 135.231,A -85,B 0,C 180,E1 -6464.143,E2 -6464.143} C_VEL
LIN {X 0,Y 488.724,Z 135.226,A -85,B 0,C 180,E1 -6466.698,E2 -6466.698} C_VEL
LIN {X 0,Y 488.735,Z 135.228,A -85,B 0,C 180,E1 -6469.226,E2 -6469.226} C_VEL
LIN {X 0,Y 488.782,Z 135.219,A -85,B 0,C 180,E1 -6471.733,E2 -6471.733} C_VEL
LIN {X 0,Y 488.84,Z 135.216,A -85,B 0,C 180,E1 -6474.224,E2 -6474.224} C_VEL
LIN {X 0,Y 488.953,Z 135.197,A -85,B 0,C 180,E1 -6477.529,E2 -6477.529} C_VEL
LIN {X 0,Y 488.97,Z 135.199,A -85,B 0,C 180,E1 -6480,E2 -6480} C_VEL
LIN {X 0,Y 488.955,Z 135.195,A -85,B 0,C 180,E1 -6482.471,E2 -6482.471} C_VEL
LIN {X 0,Y 488.842,Z 135.216,A -85,B 0,C 180,E1 -6485.776,E2 -6485.776} C_VEL
LIN {X 0,Y 488.787,Z 135.217,A -85,B 0,C 180,E1 -6488.267,E2 -6488.267} C_VEL
LIN {X 0,Y 488.808,Z 135.221,A -85,B 0,C 180,E1 -6491.612,E2 -6491.612} C_VEL
LIN {X 0,Y 488.762,Z 135.224,A -85,B 0,C 180,E1 -6495,E2 -6495} C_VEL
LIN {X 0,Y 488.747,Z 135.227,A -85,B 0,C 180,E1 -6498.442,E2 -6498.442} C_VEL
LIN {X 0,Y 488.709,Z 135.23,A -85,B 0,C 180,E1 -6501.071,E2 -6501.071} C_VEL
LIN {X 0,Y 488.673,Z 135.235,A -85,B 0,C 180,E1 -6503.746,E2 -6503.746} C_VEL
LIN {X 0,Y 488.75,Z 135.228,A -85,B 0,C 180,E1 -6506.933,E2 -6506.933} C_VEL
LIN {X 0,Y 488.724,Z 135.229,A -85,B 0,C 180,E1 -6509.27,E2 -6509.27} C_VEL
LIN {X 0,Y 488.698,Z 135.219,A -85,B 0,C 180,E1 -6512.147,E2 -6512.147} C_VEL
LIN {X 0,Y 488.716,Z 135.228,A -85,B 0,C 180,E1 -6515.115,E2 -6515.115} C_VEL
LIN {X 0,Y 488.681,Z 135.239,A -85,B 0,C 180,E1 -6518.2,E2 -6518.2} C_VEL
LIN {X 0,Y 488.719,Z 135.22,A -85,B 0,C 180,E1 -6520.344,E2 -6520.344} C_VEL
LIN {X 0,Y 488.686,Z 135.236,A -85,B 0,C 180,E1 -6523.654,E2 -6523.654} C_VEL
LIN {X 0,Y 488.685,Z 135.229,A -85,B 0,C 180,E1 -6526.345,E2 -6526.345} C_VEL
LIN {X 0,Y 488.734,Z 135.23,A -85,B 0,C 180,E1 -6529.676,E2 -6529.676} C_VEL
LIN {X 0,Y 488.68,Z 135.236,A -85,B 0,C 180,E1 -6532.841,E2 -6532.841} C_VEL
LIN {X 0,Y 488.731,Z 135.233,A -85,B 0,C 180,E1 -6535.887,E2 -6535.887} C_VEL
LIN {X 0,Y 488.692,Z 135.216,A -85,B 0,C 180,E1 -6538.82,E2 -6538.82} C_VEL
LIN {X 0,Y 488.793,Z 135.361,A -85,B 0,C 180,E1 -6541.537,E2 -6541.537} C_VEL
LIN {X 0,Y 492.251,Z 150.402,A -85,B 0,C 180,E1 -6544.088,E2 -6544.088} C_VEL
LIN {X 0,Y 492.179,Z 157.013,A -85,B 0,C 180,E1 -6545.087,E2 -6545.087} C_VEL
LIN {X 0,Y 491.614,Z 169.48,A -85,B 0,C 180,E1 -6546.906,E2 -6546.906} C_VEL
LIN {X 0,Y 495.597,Z 189.205,A -85,B 0,C 180,E1 -6547.433,E2 -6547.433} C_VEL
LIN {X 0,Y 494.177,Z 335.962,A -85,B 0,C 180,E1 -6549.636,E2 -6549.636} C_VEL
LIN {X 0,Y 493.721,Z 351.547,A -85,B 0,C 180,E1 -6550.041,E2 -6550.041} C_VEL
LIN {X 0,Y 493.22,Z 366.06,A -85,B 0,C 180,E1 -6550.583,E2 -6550.583} C_VEL
LIN {X 0,Y 492.578,Z 380.151,A -85,B 0,C 180,E1 -6551.275,E2 -6551.275} C_VEL
LIN {X 0,Y 491.92,Z 393.634,A -85,B 0,C 180,E1 -6552.111,E2 -6552.111} C_VEL
LIN {X 0,Y 491.216,Z 406.064,A -85,B 0,C 180,E1 -6553.051,E2 -6553.051} C_VEL
LIN {X 0,Y 490.623,Z 417.456,A -85,B 0,C 180,E1 -6554.082,E2 -6554.082} C_VEL
LIN {X 0,Y 489.929,Z 428.397,A -85,B 0,C 180,E1 -6555.249,E2 -6555.249} C_VEL
LIN {X 0,Y 489.408,Z 438.355,A -85,B 0,C 180,E1 -6556.505,E2 -6556.505} C_VEL
LIN {X 0,Y 488.876,Z 447.327,A -85,B 0,C 180,E1 -6557.838,E2 -6557.838} C_VEL
LIN {X 0,Y 488.631,Z 455.137,A -85,B 0,C 180,E1 -6559.223,E2 -6559.223} C_VEL
LIN {X 0,Y 488.262,Z 462.932,A -85,B 0,C 180,E1 -6560.89,E2 -6560.89} C_VEL
LIN {X 0,Y 488.073,Z 469.132,A -85,B 0,C 180,E1 -6562.554,E2 -6562.554} C_VEL
LIN {X 0,Y 488,Z 473.927,A -85,B 0,C 180,E1 -6564.214,E2 -6564.214} C_VEL
LIN {X 0,Y 487.868,Z 477.438,A -85,B 0,C 180,E1 -6565.869,E2 -6565.869} C_VEL
LIN {X 0,Y 487.882,Z 479.748,A -85,B 0,C 180,E1 -6567.523,E2 -6567.523} C_VEL
LIN {X 0,Y 487.83,Z 480.91,A -85,B 0,C 180,E1 -6569.174,E2 -6569.174} C_VEL
LIN {X 0,Y 487.83,Z 480.909,A -85,B 0,C 180,E1 -6570.825,E2 -6570.825} C_VEL
LIN {X 0,Y 487.882,Z 479.744,A -85,B 0,C 180,E1 -6572.477,E2 -6572.477} C_VEL
LIN {X 0,Y 487.868,Z 477.433,A -85,B 0,C 180,E1 -6574.13,E2 -6574.13} C_VEL
LIN {X 0,Y 488.01,Z 473.928,A -85,B 0,C 180,E1 -6575.786,E2 -6575.786} C_VEL
LIN {X 0,Y 488.073,Z 469.137,A -85,B 0,C 180,E1 -6577.446,E2 -6577.446} C_VEL
LIN {X 0,Y 488.262,Z 462.929,A -85,B 0,C 180,E1 -6579.11,E2 -6579.11} C_VEL
LIN {X 0,Y 488.635,Z 455.131,A -85,B 0,C 180,E1 -6580.776,E2 -6580.776} C_VEL
LIN {X 0,Y 488.904,Z 447.232,A -85,B 0,C 180,E1 -6582.177,E2 -6582.177} C_VEL
LIN {X 0,Y 489.506,Z 436.839,A -85,B 0,C 180,E1 -6583.703,E2 -6583.703} C_VEL
LIN {X 0,Y 490.032,Z 426.61,A -85,B 0,C 180,E1 -6584.961,E2 -6584.961} C_VEL
LIN {X 0,Y 490.718,Z 414.513,A -85,B 0,C 180,E1 -6586.208,E2 -6586.208} C_VEL
LIN {X 0,Y 491.427,Z 402.187,A -85,B 0,C 180,E1 -6587.263,E2 -6587.263} C_VEL
LIN {X 0,Y 492.145,Z 388.87,A -85,B 0,C 180,E1 -6588.203,E2 -6588.203} C_VEL
LIN {X 0,Y 492.756,Z 376.157,A -85,B 0,C 180,E1 -6588.934,E2 -6588.934} C_VEL
LIN {X 0,Y 493.362,Z 361.482,A -85,B 0,C 180,E1 -6589.602,E2 -6589.602} C_VEL
LIN {X 0,Y 493.882,Z 346.481,A -85,B 0,C 180,E1 -6590.106,E2 -6590.106} C_VEL
LIN {X 0,Y 494.193,Z 332.002,A -85,B 0,C 180,E1 -6590.437,E2 -6590.437} C_VEL
LIN {X 0,Y 495.609,Z 189.44,A -85,B 0,C 180,E1 -6592.561,E2 -6592.561} C_VEL
LIN {X 0,Y 491.621,Z 169.74,A -85,B 0,C 180,E1 -6593.074,E2 -6593.074} C_VEL
LIN {X 0,Y 492.311,Z 154.021,A -85,B 0,C 180,E1 -6595.358,E2 -6595.358} C_VEL
LIN {X 0,Y 492.241,Z 150.415,A -85,B 0,C 180,E1 -6595.91,E2 -6595.91} C_VEL
LIN {X 0,Y 488.81,Z 135.536,A -85,B 0,C 180,E1 -6598.416,E2 -6598.416} C_VEL
LIN {X 0,Y 488.731,Z 135.214,A -85,B 0,C 180,E1 -6598.696,E2 -6598.696} C_VEL
LIN {X 0,Y 488.692,Z 135.216,A -85,B 0,C 180,E1 -6601.18,E2 -6601.18} C_VEL
LIN {X 0,Y 488.731,Z 135.233,A -85,B 0,C 180,E1 -6604.113,E2 -6604.113} C_VEL
LIN {X 0,Y 488.68,Z 135.235,A -85,B 0,C 180,E1 -6607.159,E2 -6607.159} C_VEL
LIN {X 0,Y 488.719,Z 135.233,A -85,B 0,C 180,E1 -6610.345,E2 -6610.345} C_VEL
LIN {X 0,Y 488.684,Z 135.229,A -85,B 0,C 180,E1 -6613.655,E2 -6613.655} C_VEL
LIN {X 0,Y 488.685,Z 135.236,A -85,B 0,C 180,E1 -6616.346,E2 -6616.346} C_VEL
LIN {X 0,Y 488.734,Z 135.218,A -85,B 0,C 180,E1 -6619.677,E2 -6619.677} C_VEL
LIN {X 0,Y 488.68,Z 135.235,A -85,B 0,C 180,E1 -6622.841,E2 -6622.841} C_VEL
LIN {X 0,Y 488.721,Z 135.213,A -85,B 0,C 180,E1 -6625.887,E2 -6625.887} C_VEL
LIN {X 0,Y 488.691,Z 135.223,A -85,B 0,C 180,E1 -6628.82,E2 -6628.82} C_VEL
LIN {X 0,Y 488.745,Z 135.229,A -85,B 0,C 180,E1 -6631.671,E2 -6631.671} C_VEL
LIN {X 0,Y 488.74,Z 135.222,A -85,B 0,C 180,E1 -6634.444,E2 -6634.444} C_VEL
LIN {X 0,Y 488.724,Z 135.233,A -85,B 0,C 180,E1 -6637.153,E2 -6637.153} C_VEL
LIN {X 0,Y 488.725,Z 135.226,A -85,B 0,C 180,E1 -6639.811,E2 -6639.811} C_VEL
LIN {X 0,Y 488.711,Z 135.232,A -85,B 0,C 180,E1 -6642.423,E2 -6642.423} C_VEL
LIN {X 0,Y 488.762,Z 135.223,A -85,B 0,C 180,E1 -6645,E2 -6645} C_VEL
LIN {X 0,Y 488.807,Z 135.221,A -85,B 0,C 180,E1 -6648.388,E2 -6648.388} C_VEL
LIN {X 0,Y 488.787,Z 135.217,A -85,B 0,C 180,E1 -6651.733,E2 -6651.733} C_VEL
LIN {X 0,Y 488.843,Z 135.216,A -85,B 0,C 180,E1 -6654.224,E2 -6654.224} C_VEL
LIN {X 0,Y 488.956,Z 135.195,A -85,B 0,C 180,E1 -6657.529,E2 -6657.529} C_VEL
LIN {X 0,Y 488.915,Z 135.203,A -85,B 0,C 180,E1 -6660.824,E2 -6660.824} C_VEL
LIN {X 0,Y 488.953,Z 135.197,A -85,B 0,C 180,E1 -6662.471,E2 -6662.471} C_VEL
LIN {X 0,Y 488.84,Z 135.215,A -85,B 0,C 180,E1 -6665.776,E2 -6665.776} C_VEL
LIN {X 0,Y 488.787,Z 135.219,A -85,B 0,C 180,E1 -6668.267,E2 -6668.267} C_VEL
LIN {X 0,Y 488.807,Z 135.22,A -85,B 0,C 180,E1 -6671.612,E2 -6671.612} C_VEL
LIN {X 0,Y 488.751,Z 135.219,A -85,B 0,C 180,E1 -6675.001,E2 -6675.001} C_VEL
LIN {X 0,Y 488.746,Z 135.225,A -85,B 0,C 180,E1 -6678.443,E2 -6678.443} C_VEL
LIN {X 0,Y 488.708,Z 135.227,A -85,B 0,C 180,E1 -6681.071,E2 -6681.071} C_VEL
LIN {X 0,Y 488.671,Z 135.24,A -85,B 0,C 180,E1 -6683.747,E2 -6683.747} C_VEL
LIN {X 0,Y 488.699,Z 135.231,A -85,B 0,C 180,E1 -6686.922,E2 -6686.922} C_VEL
LIN {X 0,Y 488.719,Z 135.22,A -85,B 0,C 180,E1 -6690.22,E2 -6690.22} C_VEL
LIN {X 0,Y 488.711,Z 135.216,A -85,B 0,C 180,E1 -6693.48,E2 -6693.48} C_VEL
LIN {X 0,Y 488.673,Z 135.236,A -85,B 0,C 180,E1 -6696.353,E2 -6696.353} C_VEL
LIN {X 0,Y 488.694,Z 135.223,A -85,B 0,C 180,E1 -6699.255,E2 -6699.255} C_VEL
LIN {X 0,Y 488.668,Z 135.233,A -85,B 0,C 180,E1 -6701.594,E2 -6701.594} C_VEL
LIN {X 0,Y 488.702,Z 135.234,A -85,B 0,C 180,E1 -6704.803,E2 -6704.803} C_VEL
LIN {X 0,Y 488.65,Z 135.243,A -85,B 0,C 180,E1 -6707.47,E2 -6707.47} C_VEL
LIN {X 0,Y 488.704,Z 135.226,A -85,B 0,C 180,E1 -6709.674,E2 -6709.674} C_VEL
LIN {X 0,Y 488.668,Z 135.24,A -85,B 0,C 180,E1 -6712.84,E2 -6712.84} C_VEL
LIN {X 0,Y 488.721,Z 135.229,A -85,B 0,C 180,E1 -6715.886,E2 -6715.886} C_VEL
LIN {X 0,Y 488.662,Z 135.229,A -85,B 0,C 180,E1 -6718.818,E2 -6718.818} C_VEL
LIN {X 0,Y 488.681,Z 135.232,A -85,B 0,C 180,E1 -6722.134,E2 -6722.134} C_VEL
LIN {X 0,Y 488.766,Z 135.497,A -85,B 0,C 180,E1 -6722.67,E2 -6722.67} C_VEL
LIN {X 0,Y 489.239,Z 137.632,A -85,B 0,C 180,E1 -6723.071,E2 -6723.071} C_VEL
LIN {X 0,Y 489.377,Z 141.057,A -85,B 0,C 180,E1 -6723.636,E2 -6723.636} C_VEL
LIN {X 0,Y 487.824,Z 147.176,A -85,B 0,C 180,E1 -6724.534,E2 -6724.534} C_VEL
LIN {X 0,Y 486.104,Z 152.208,A -85,B 0,C 180,E1 -6725.246,E2 -6725.246} C_VEL
LIN {X 0,Y 485.083,Z 157.152,A -85,B 0,C 180,E1 -6725.983,E2 -6725.983} C_VEL
LIN {X 0,Y 484.907,Z 161.638,A -85,B 0,C 180,E1 -6726.638,E2 -6726.638} C_VEL
LIN {X 0,Y 489.09,Z 181.27,A -85,B 0,C 180,E1 -6727.171,E2 -6727.171} C_VEL
LIN {X 0,Y 487.593,Z 327.152,A -85,B 0,C 180,E1 -6729.39,E2 -6729.39} C_VEL
LIN {X 0,Y 487.128,Z 342.655,A -85,B 0,C 180,E1 -6729.794,E2 -6729.794} C_VEL
LIN {X 0,Y 486.688,Z 357.271,A -85,B 0,C 180,E1 -6730.35,E2 -6730.35} C_VEL
LIN {X 0,Y 485.984,Z 370.658,A -85,B 0,C 180,E1 -6731.011,E2 -6731.011} C_VEL
LIN {X 0,Y 485.296,Z 384.283,A -85,B 0,C 180,E1 -6731.859,E2 -6731.859} C_VEL
LIN {X 0,Y 484.519,Z 396.814,A -85,B 0,C 180,E1 -6732.81,E2 -6732.81} C_VEL
LIN {X 0,Y 483.776,Z 409.503,A -85,B 0,C 180,E1 -6733.977,E2 -6733.977} C_VEL
LIN {X 0,Y 483.057,Z 421.01,A -85,B 0,C 180,E1 -6735.25,E2 -6735.25} C_VEL
LIN {X 0,Y 482.483,Z 430.694,A -85,B 0,C 180,E1 -6736.523,E2 -6736.523} C_VEL
LIN {X 0,Y 481.924,Z 440.28,A -85,B 0,C 180,E1 -6738.022,E2 -6738.022} C_VEL
LIN {X 0,Y 481.546,Z 448.093,A -85,B 0,C 180,E1 -6739.488,E2 -6739.488} C_VEL
LIN {X 0,Y 481.212,Z 455.476,A -85,B 0,C 180,E1 -6741.179,E2 -6741.179} C_VEL
LIN {X 0,Y 480.996,Z 461.336,A -85,B 0,C 180,E1 -6742.866,E2 -6742.866} C_VEL
LIN {X 0,Y 480.973,Z 464.806,A -85,B 0,C 180,E1 -6744.129,E2 -6744.129} C_VEL
LIN {X 0,Y 480.802,Z 468.327,A -85,B 0,C 180,E1 -6745.809,E2 -6745.809} C_VEL
LIN {X 0,Y 480.819,Z 470.656,A -85,B 0,C 180,E1 -6747.487,E2 -6747.487} C_VEL
LIN {X 0,Y 480.757,Z 471.85,A -85,B 0,C 180,E1 -6749.162,E2 -6749.162} C_VEL
LIN {X 0,Y 480.757,Z 471.868,A -85,B 0,C 180,E1 -6750.838,E2 -6750.838} C_VEL
LIN {X 0,Y 480.82,Z 470.746,A -85,B 0,C 180,E1 -6752.513,E2 -6752.513} C_VEL
LIN {X 0,Y 480.802,Z 468.487,A -85,B 0,C 180,E1 -6754.191,E2 -6754.191} C_VEL
LIN {X 0,Y 480.951,Z 465.032,A -85,B 0,C 180,E1 -6755.871,E2 -6755.871} C_VEL
LIN {X 0,Y 481.036,Z 460.305,A -85,B 0,C 180,E1 -6757.556,E2 -6757.556} C_VEL
LIN {X 0,Y 481.265,Z 454.179,A -85,B 0,C 180,E1 -6759.244,E2 -6759.244} C_VEL
LIN {X 0,Y 481.727,Z 446.467,A -85,B 0,C 180,E1 -6760.933,E2 -6760.933} C_VEL
LIN {X 0,Y 482.025,Z 438.671,A -85,B 0,C 180,E1 -6762.346,E2 -6762.346} C_VEL
LIN {X 0,Y 482.645,Z 428.349,A -85,B 0,C 180,E1 -6763.902,E2 -6763.902} C_VEL
LIN {X 0,Y 483.261,Z 418.201,A -85,B 0,C 180,E1 -6765.175,E2 -6765.175} C_VEL
LIN {X 0,Y 484.004,Z 406.269,A -85,B 0,C 180,E1 -6766.433,E2 -6766.433} C_VEL
LIN {X 0,Y 484.719,Z 394.017,A -85,B 0,C 180,E1 -6767.509,E2 -6767.509} C_VEL
LIN {X 0,Y 485.473,Z 380.867,A -85,B 0,C 180,E1 -6768.462,E2 -6768.462} C_VEL
LIN {X 0,Y 486.091,Z 368.346,A -85,B 0,C 180,E1 -6769.204,E2 -6769.204} C_VEL
LIN {X 0,Y 486.816,Z 353.09,A -85,B 0,C 180,E1 -6769.913,E2 -6769.913} C_VEL
LIN {X 0,Y 487.237,Z 338.977,A -85,B 0,C 180,E1 -6770.405,E2 -6770.405} C_VEL
LIN {X 0,Y 487.622,Z 323.443,A -85,B 0,C 180,E1 -6770.77,E2 -6770.77} C_VEL
LIN {X 0,Y 489.095,Z 182.012,A -85,B 0,C 180,E1 -6772.909,E2 -6772.909} C_VEL
LIN {X 0,Y 485.502,Z 164.251,A -85,B 0,C 180,E1 -6773.369,E2 -6773.369} C_VEL
LIN {X 0,Y 484.912,Z 161.195,A -85,B 0,C 180,E1 -6773.489,E2 -6773.489} C_VEL
LIN {X 0,Y 485.28,Z 152.58,A -85,B 0,C 180,E1 -6774.834,E2 -6774.834} C_VEL
LIN {X 0,Y 482.063,Z 137.926,A -85,B 0,C 180,E1 -6777.419,E2 -6777.419} C_VEL
LIN {X 0,Y 481.654,Z 136.159,A -85,B 0,C 180,E1 -6777.81,E2 -6777.81} C_VEL
LIN {X 0,Y 481.609,Z 136.099,A -85,B 0,C 180,E1 -6780.714,E2 -6780.714} C_VEL
LIN {X 0,Y 481.676,Z 136.107,A -85,B 0,C 180,E1 -6783.729,E2 -6783.729} C_VEL
LIN {X 0,Y 481.608,Z 136.114,A -85,B 0,C 180,E1 -6786.749,E2 -6786.749} C_VEL
LIN {X 0,Y 481.656,Z 136.102,A -85,B 0,C 180,E1 -6789.943,E2 -6789.943} C_VEL
LIN {X 0,Y 481.619,Z 136.109,A -85,B 0,C 180,E1 -6793.302,E2 -6793.302} C_VEL
LIN {X 0,Y 481.653,Z 136.109,A -85,B 0,C 180,E1 -6795.642,E2 -6795.642} C_VEL
LIN {X 0,Y 481.623,Z 136.101,A -85,B 0,C 180,E1 -6798.955,E2 -6798.955} C_VEL
LIN {X 0,Y 481.639,Z 136.106,A -85,B 0,C 180,E1 -6801.995,E2 -6801.995} C_VEL
LIN {X 0,Y 481.682,Z 136.102,A -85,B 0,C 180,E1 -6805.317,E2 -6805.317} C_VEL
LIN {X 0,Y 481.643,Z 136.09,A -85,B 0,C 180,E1 -6808.311,E2 -6808.311} C_VEL
LIN {X 0,Y 481.661,Z 136.108,A -85,B 0,C 180,E1 -6811.216,E2 -6811.216} C_VEL
LIN {X 0,Y 481.644,Z 136.114,A -85,B 0,C 180,E1 -6814.039,E2 -6814.039} C_VEL
LIN {X 0,Y 481.676,Z 136.108,A -85,B 0,C 180,E1 -6816.812,E2 -6816.812} C_VEL
LIN {X 0,Y 481.695,Z 136.102,A -85,B 0,C 180,E1 -6819.503,E2 -6819.503} C_VEL
LIN {X 0,Y 481.673,Z 136.114,A -85,B 0,C 180,E1 -6822.157,E2 -6822.157} C_VEL
LIN {X 0,Y 481.732,Z 136.094,A -85,B 0,C 180,E1 -6824.775,E2 -6824.775} C_VEL
LIN {X 0,Y 481.753,Z 136.101,A -85,B 0,C 180,E1 -6828.215,E2 -6828.215} C_VEL
LIN {X 0,Y 481.738,Z 136.096,A -85,B 0,C 180,E1 -6831.611,E2 -6831.611} C_VEL
LIN {X 0,Y 481.799,Z 136.094,A -85,B 0,C 180,E1 -6834.139,E2 -6834.139} C_VEL
LIN {X 0,Y 481.918,Z 136.073,A -85,B 0,C 180,E1 -6837.492,E2 -6837.492} C_VEL
LIN {X 0,Y 481.941,Z 136.075,A -85,B 0,C 180,E1 -6840,E2 -6840} C_VEL
LIN {X 0,Y 481.922,Z 136.071,A -85,B 0,C 180,E1 -6842.507,E2 -6842.507} C_VEL
LIN {X 0,Y 481.801,Z 136.092,A -85,B 0,C 180,E1 -6845.861,E2 -6845.861} C_VEL
LIN {X 0,Y 481.742,Z 136.095,A -85,B 0,C 180,E1 -6848.389,E2 -6848.389} C_VEL
LIN {X 0,Y 481.753,Z 136.098,A -85,B 0,C 180,E1 -6851.785,E2 -6851.785} C_VEL
LIN {X 0,Y 481.744,Z 136.096,A -85,B 0,C 180,E1 -6855.224,E2 -6855.224} C_VEL
LIN {X 0,Y 481.709,Z 136.107,A -85,B 0,C 180,E1 -6858.722,E2 -6858.722} C_VEL
LIN {X 0,Y 481.647,Z 136.109,A -85,B 0,C 180,E1 -6861.395,E2 -6861.395} C_VEL
LIN {X 0,Y 481.652,Z 136.11,A -85,B 0,C 180,E1 -6864.114,E2 -6864.114} C_VEL
LIN {X 0,Y 481.717,Z 136.104,A -85,B 0,C 180,E1 -6867.132,E2 -6867.132} C_VEL
LIN {X 0,Y 481.68,Z 136.105,A -85,B 0,C 180,E1 -6869.741,E2 -6869.741} C_VEL
LIN {X 0,Y 481.653,Z 136.09,A -85,B 0,C 180,E1 -6872.676,E2 -6872.676} C_VEL
LIN {X 0,Y 481.637,Z 136.109,A -85,B 0,C 180,E1 -6875.709,E2 -6875.709} C_VEL
LIN {X 0,Y 481.671,Z 136.101,A -85,B 0,C 180,E1 -6878.859,E2 -6878.859} C_VEL
LIN {X 0,Y 481.653,Z 136.105,A -85,B 0,C 180,E1 -6881.913,E2 -6881.913} C_VEL
LIN {X 0,Y 481.656,Z 136.109,A -85,B 0,C 180,E1 -6884.458,E2 -6884.458} C_VEL
LIN {X 0,Y 481.648,Z 136.112,A -85,B 0,C 180,E1 -6887.839,E2 -6887.839} C_VEL
LIN {X 0,Y 481.663,Z 136.105,A -85,B 0,C 180,E1 -6890.654,E2 -6890.654} C_VEL
LIN {X 0,Y 481.628,Z 136.115,A -85,B 0,C 180,E1 -6893.376,E2 -6893.376} C_VEL
LIN {X 0,Y 481.71,Z 136.1,A -85,B 0,C 180,E1 -6896.33,E2 -6896.33} C_VEL
LIN {X 0,Y 481.651,Z 136.101,A -85,B 0,C 180,E1 -6899.417,E2 -6899.417} C_VEL
LIN {X 0,Y 481.737,Z 136.3,A -85,B 0,C 180,E1 -6901.251,E2 -6901.251} C_VEL
LIN {X 0,Y 485.293,Z 151.583,A -85,B 0,C 180,E1 -6903.881,E2 -6903.881} C_VEL
LIN {X 0,Y 485.496,Z 155.459,A -85,B 0,C 180,E1 -6904.491,E2 -6904.491} C_VEL
LIN {X 0,Y 484.839,Z 169.408,A -85,B 0,C 180,E1 -6906.564,E2 -6906.564} C_VEL
LIN {X 0,Y 488.602,Z 188.047,A -85,B 0,C 180,E1 -6907.075,E2 -6907.075} C_VEL
LIN {X 0,Y 489.01,Z 190.761,A -85,B 0,C 180,E1 -6907.137,E2 -6907.137} C_VEL
LIN {X 0,Y 487.536,Z 334.576,A -85,B 0,C 180,E1 -6909.319,E2 -6909.319} C_VEL
LIN {X 0,Y 487.074,Z 350.22,A -85,B 0,C 180,E1 -6909.714,E2 -6909.714} C_VEL
LIN {X 0,Y 486.538,Z 365.247,A -85,B 0,C 180,E1 -6910.273,E2 -6910.273} C_VEL
LIN {X 0,Y 485.854,Z 380.089,A -85,B 0,C 180,E1 -6911.006,E2 -6911.006} C_VEL
LIN {X 0,Y 485.142,Z 393.571,A -85,B 0,C 180,E1 -6911.853,E2 -6911.853} C_VEL
LIN {X 0,Y 484.376,Z 406,A -85,B 0,C 180,E1 -6912.805,E2 -6912.805} C_VEL
LIN {X 0,Y 483.753,Z 416.889,A -85,B 0,C 180,E1 -6913.799,E2 -6913.799} C_VEL
LIN {X 0,Y 483.003,Z 428.331,A -85,B 0,C 180,E1 -6915.032,E2 -6915.032} C_VEL
LIN {X 0,Y 482.462,Z 438.289,A -85,B 0,C 180,E1 -6916.307,E2 -6916.307} C_VEL
LIN {X 0,Y 481.851,Z 447.781,A -85,B 0,C 180,E1 -6917.748,E2 -6917.748} C_VEL
LIN {X 0,Y 481.565,Z 456.153,A -85,B 0,C 180,E1 -6919.276,E2 -6919.276} C_VEL
LIN {X 0,Y 481.207,Z 462.866,A -85,B 0,C 180,E1 -6920.755,E2 -6920.755} C_VEL
LIN {X 0,Y 480.996,Z 469.066,A -85,B 0,C 180,E1 -6922.444,E2 -6922.444} C_VEL
LIN {X 0,Y 480.904,Z 473.86,A -85,B 0,C 180,E1 -6924.128,E2 -6924.128} C_VEL
LIN {X 0,Y 480.775,Z 477.371,A -85,B 0,C 180,E1 -6925.808,E2 -6925.808} C_VEL
LIN {X 0,Y 480.798,Z 479.682,A -85,B 0,C 180,E1 -6927.487,E2 -6927.487} C_VEL
LIN {X 0,Y 480.756,Z 480.844,A -85,B 0,C 180,E1 -6929.162,E2 -6929.162} C_VEL
LIN {X 0,Y 480.756,Z 480.843,A -85,B 0,C 180,E1 -6930.838,E2 -6930.838} C_VEL
LIN {X 0,Y 480.798,Z 479.678,A -85,B 0,C 180,E1 -6932.513,E2 -6932.513} C_VEL
LIN {X 0,Y 480.775,Z 477.367,A -85,B 0,C 180,E1 -6934.191,E2 -6934.191} C_VEL
LIN {X 0,Y 480.919,Z 473.862,A -85,B 0,C 180,E1 -6935.871,E2 -6935.871} C_VEL
LIN {X 0,Y 480.997,Z 469.069,A -85,B 0,C 180,E1 -6937.556,E2 -6937.556} C_VEL
LIN {X 0,Y 481.207,Z 462.862,A -85,B 0,C 180,E1 -6939.245,E2 -6939.245} C_VEL
LIN {X 0,Y 481.613,Z 455.064,A -85,B 0,C 180,E1 -6940.936,E2 -6940.936} C_VEL
LIN {X 0,Y 481.921,Z 447.141,A -85,B 0,C 180,E1 -6942.36,E2 -6942.36} C_VEL
LIN {X 0,Y 482.556,Z 436.771,A -85,B 0,C 180,E1 -6943.905,E2 -6943.905} C_VEL
LIN {X 0,Y 483.115,Z 426.542,A -85,B 0,C 180,E1 -6945.18,E2 -6945.18} C_VEL
LIN {X 0,Y 483.849,Z 414.444,A -85,B 0,C 180,E1 -6946.445,E2 -6946.445} C_VEL
LIN {X 0,Y 484.6,Z 402.118,A -85,B 0,C 180,E1 -6947.514,E2 -6947.514} C_VEL
LIN {X 0,Y 485.357,Z 388.8,A -85,B 0,C 180,E1 -6948.467,E2 -6948.467} C_VEL
LIN {X 0,Y 486.038,Z 376.087,A -85,B 0,C 180,E1 -6949.206,E2 -6949.206} C_VEL
LIN {X 0,Y 486.648,Z 362.038,A -85,B 0,C 180,E1 -6949.858,E2 -6949.858} C_VEL
LIN {X 0,Y 487.209,Z 346.901,A -85,B 0,C 180,E1 -6950.379,E2 -6950.379} C_VEL
LIN {X 0,Y 487.58,Z 331.492,A -85,B 0,C 180,E1 -6950.735,E2 -6950.735} C_VEL
LIN {X 0,Y 489.05,Z 190.662,A -85,B 0,C 180,E1 -6952.861,E2 -6952.861} C_VEL
LIN {X 0,Y 484.833,Z 169.654,A -85,B 0,C 180,E1 -6953.417,E2 -6953.417} C_VEL
LIN {X 0,Y 485.556,Z 153.957,A -85,B 0,C 180,E1 -6955.736,E2 -6955.736} C_VEL
LIN {X 0,Y 484.247,Z 146.754,A -85,B 0,C 180,E1 -6956.928,E2 -6956.928} C_VEL
LIN {X 0,Y 481.7,Z 136.202,A -85,B 0,C 180,E1 -6958.781,E2 -6958.781} C_VEL
LIN {X 0,Y 481.657,Z 136.089,A -85,B 0,C 180,E1 -6962.189,E2 -6962.189} C_VEL
LIN {X 0,Y 481.689,Z 136.108,A -85,B 0,C 180,E1 -6964.682,E2 -6964.682} C_VEL
LIN {X 0,Y 481.656,Z 136.114,A -85,B 0,C 180,E1 -6968.007,E2 -6968.007} C_VEL
LIN {X 0,Y 481.656,Z 136.11,A -85,B 0,C 180,E1 -6971.042,E2 -6971.042} C_VEL
LIN {X 0,Y 481.655,Z 136.105,A -85,B 0,C 180,E1 -6974.458,E2 -6974.458} C_VEL
LIN {X 0,Y 481.648,Z 136.108,A -85,B 0,C 180,E1 -6977.839,E2 -6977.839} C_VEL
LIN {X 0,Y 481.68,Z 136.098,A -85,B 0,C 180,E1 -6980.651,E2 -6980.651} C_VEL
LIN {X 0,Y 481.628,Z 136.119,A -85,B 0,C 180,E1 -6983.376,E2 -6983.376} C_VEL
LIN {X 0,Y 481.67,Z 136.088,A -85,B 0,C 180,E1 -6986.327,E2 -6986.327} C_VEL
LIN {X 0,Y 481.65,Z 136.107,A -85,B 0,C 180,E1 -6989.418,E2 -6989.418} C_VEL
LIN {X 0,Y 481.7,Z 136.103,A -85,B 0,C 180,E1 -6992.168,E2 -6992.168} C_VEL
LIN {X 0,Y 481.713,Z 136.101,A -85,B 0,C 180,E1 -6994.97,E2 -6994.97} C_VEL
LIN {X 0,Y 481.65,Z 136.107,A -85,B 0,C 180,E1 -6997.705,E2 -6997.705} C_VEL
LIN {X 0,Y 481.704,Z 136.101,A -85,B 0,C 180,E1 -7000.393,E2 -7000.393} C_VEL
LIN {X 0,Y 481.675,Z 136.108,A -85,B 0,C 180,E1 -7003.033,E2 -7003.033} C_VEL
LIN {X 0,Y 481.688,Z 136.104,A -85,B 0,C 180,E1 -7005.639,E2 -7005.639} C_VEL
LIN {X 0,Y 481.753,Z 136.098,A -85,B 0,C 180,E1 -7008.215,E2 -7008.215} C_VEL
LIN {X 0,Y 481.741,Z 136.095,A -85,B 0,C 180,E1 -7011.611,E2 -7011.611} C_VEL
LIN {X 0,Y 481.801,Z 136.092,A -85,B 0,C 180,E1 -7014.139,E2 -7014.139} C_VEL
LIN {X 0,Y 481.922,Z 136.071,A -85,B 0,C 180,E1 -7017.493,E2 -7017.493} C_VEL
LIN {X 0,Y 481.941,Z 136.075,A -85,B 0,C 180,E1 -7020,E2 -7020} C_VEL
LIN {X 0,Y 481.919,Z 136.073,A -85,B 0,C 180,E1 -7022.508,E2 -7022.508} C_VEL
LIN {X 0,Y 481.799,Z 136.093,A -85,B 0,C 180,E1 -7025.861,E2 -7025.861} C_VEL
LIN {X 0,Y 481.742,Z 136.095,A -85,B 0,C 180,E1 -7028.389,E2 -7028.389} C_VEL
LIN {X 0,Y 481.753,Z 136.1,A -85,B 0,C 180,E1 -7031.785,E2 -7031.785} C_VEL
LIN {X 0,Y 481.732,Z 136.094,A -85,B 0,C 180,E1 -7035.225,E2 -7035.225} C_VEL
LIN {X 0,Y 481.707,Z 136.1,A -85,B 0,C 180,E1 -7038.722,E2 -7038.722} C_VEL
LIN {X 0,Y 481.646,Z 136.108,A -85,B 0,C 180,E1 -7041.395,E2 -7041.395} C_VEL
LIN {X 0,Y 481.649,Z 136.109,A -85,B 0,C 180,E1 -7044.115,E2 -7044.115} C_VEL
LIN {X 0,Y 481.654,Z 136.11,A -85,B 0,C 180,E1 -7047.117,E2 -7047.117} C_VEL
LIN {X 0,Y 481.667,Z 136.104,A -85,B 0,C 180,E1 -7049.742,E2 -7049.742} C_VEL
LIN {X 0,Y 481.653,Z 136.087,A -85,B 0,C 180,E1 -7052.676,E2 -7052.676} C_VEL
LIN {X 0,Y 481.631,Z 136.118,A -85,B 0,C 180,E1 -7055.71,E2 -7055.71} C_VEL
LIN {X 0,Y 481.666,Z 136.104,A -85,B 0,C 180,E1 -7058.86,E2 -7058.86} C_VEL
LIN {X 0,Y 481.616,Z 136.112,A -85,B 0,C 180,E1 -7062.164,E2 -7062.164} C_VEL
LIN {X 0,Y 481.654,Z 136.11,A -85,B 0,C 180,E1 -7064.458,E2 -7064.458} C_VEL
LIN {X 0,Y 481.616,Z 136.11,A -85,B 0,C 180,E1 -7066.855,E2 -7066.855} C_VEL
LIN {X 0,Y 481.657,Z 136.102,A -85,B 0,C 180,E1 -7070.058,E2 -7070.058} C_VEL
LIN {X 0,Y 481.619,Z 136.113,A -85,B 0,C 180,E1 -7073.252,E2 -7073.252} C_VEL
LIN {X 0,Y 481.671,Z 136.108,A -85,B 0,C 180,E1 -7076.327,E2 -7076.327} C_VEL
LIN {X 0,Y 481.611,Z 136.099,A -85,B 0,C 180,E1 -7079.426,E2 -7079.426} C_VEL
LIN {X 0,Y 481.698,Z 136.304,A -85,B 0,C 180,E1 -7082.352,E2 -7082.352} C_VEL
LIN {X 0,Y 484.973,Z 150.581,A -85,B 0,C 180,E1 -7084.92,E2 -7084.92} C_VEL
LIN {X 0,Y 485.207,Z 154.737,A -85,B 0,C 180,E1 -7085.602,E2 -7085.602} C_VEL
LIN {X 0,Y 485.083,Z 157.152,A -85,B 0,C 180,E1 -7085.983,E2 -7085.983} C_VEL
LIN {X 0,Y 484.855,Z 160.384,A -85,B 0,C 180,E1 -7086.325,E2 -7086.325} C_VEL
LIN {X 0,Y 484.453,Z 165.434,A -85,B 0,C 180,E1 -7086.588,E2 -7086.588} C_VEL
LIN {X 0,Y 483.721,Z 173.222,A -85,B 0,C 180,E1 -7086.775,E2 -7086.775} C_VEL
LIN {X 0,Y 482.597,Z 182.181,A -85,B 0,C 180,E1 -7086.858,E2 -7086.858} C_VEL
LIN {X 0,Y 482.481,Z 187.574,A -85,B 0,C 180,E1 -7086.939,E2 -7086.939} C_VEL
LIN {X 0,Y 480.96,Z 327.238,A -85,B 0,C 180,E1 -7089.092,E2 -7089.092} C_VEL
LIN {X 0,Y 480.482,Z 342.734,A -85,B 0,C 180,E1 -7089.502,E2 -7089.502} C_VEL
LIN {X 0,Y 479.99,Z 357.57,A -85,B 0,C 180,E1 -7090.075,E2 -7090.075} C_VEL
LIN {X 0,Y 479.155,Z 372.632,A -85,B 0,C 180,E1 -7090.841,E2 -7090.841} C_VEL
LIN {X 0,Y 478.427,Z 385.923,A -85,B 0,C 180,E1 -7091.7,E2 -7091.7} C_VEL
LIN {X 0,Y 477.584,Z 399.435,A -85,B 0,C 180,E1 -7092.773,E2 -7092.773} C_VEL
LIN {X 0,Y 476.763,Z 411.691,A -85,B 0,C 180,E1 -7093.955,E2 -7093.955} C_VEL
LIN {X 0,Y 476.064,Z 422.855,A -85,B 0,C 180,E1 -7095.247,E2 -7095.247} C_VEL
LIN {X 0,Y 475.332,Z 433.705,A -85,B 0,C 180,E1 -7096.752,E2 -7096.752} C_VEL
LIN {X 0,Y 474.872,Z 442.707,A -85,B 0,C 180,E1 -7098.258,E2 -7098.258} C_VEL
LIN {X 0,Y 474.397,Z 450.172,A -85,B 0,C 180,E1 -7099.76,E2 -7099.76} C_VEL
LIN {X 0,Y 474.101,Z 457.153,A -85,B 0,C 180,E1 -7101.475,E2 -7101.475} C_VEL
LIN {X 0,Y 473.906,Z 462.641,A -85,B 0,C 180,E1 -7103.186,E2 -7103.186} C_VEL
LIN {X 0,Y 473.803,Z 466.787,A -85,B 0,C 180,E1 -7104.894,E2 -7104.894} C_VEL
LIN {X 0,Y 473.78,Z 469.703,A -85,B 0,C 180,E1 -7106.598,E2 -7106.598} C_VEL
LIN {X 0,Y 473.695,Z 471.46,A -85,B 0,C 180,E1 -7108.3,E2 -7108.3} C_VEL
LIN {X 0,Y 473.668,Z 472.075,A -85,B 0,C 180,E1 -7110,E2 -7110} C_VEL
LIN {X 0,Y 473.696,Z 471.513,A -85,B 0,C 180,E1 -7111.7,E2 -7111.7} C_VEL
LIN {X 0,Y 473.78,Z 469.827,A -85,B 0,C 180,E1 -7113.402,E2 -7113.402} C_VEL
LIN {X 0,Y 473.797,Z 466.978,A -85,B 0,C 180,E1 -7115.106,E2 -7115.106} C_VEL
LIN {X 0,Y 473.891,Z 462.899,A -85,B 0,C 180,E1 -7116.814,E2 -7116.814} C_VEL
LIN {X 0,Y 474.091,Z 457.491,A -85,B 0,C 180,E1 -7118.525,E2 -7118.525} C_VEL
LIN {X 0,Y 474.378,Z 450.602,A -85,B 0,C 180,E1 -7120.241,E2 -7120.241} C_VEL
LIN {X 0,Y 474.797,Z 443.192,A -85,B 0,C 180,E1 -7121.743,E2 -7121.743} C_VEL
LIN {X 0,Y 475.291,Z 434.27,A -85,B 0,C 180,E1 -7123.25,E2 -7123.25} C_VEL
LIN {X 0,Y 475.882,Z 425.175,A -85,B 0,C 180,E1 -7124.54,E2 -7124.54} C_VEL
LIN {X 0,Y 476.558,Z 414.448,A -85,B 0,C 180,E1 -7125.833,E2 -7125.833} C_VEL
LIN {X 0,Y 477.329,Z 403.247,A -85,B 0,C 180,E1 -7126.968,E2 -7126.968} C_VEL
LIN {X 0,Y 478.188,Z 389.959,A -85,B 0,C 180,E1 -7128.088,E2 -7128.088} C_VEL
LIN {X 0,Y 479.005,Z 375.858,A -85,B 0,C 180,E1 -7129.054,E2 -7129.054} C_VEL
LIN {X 0,Y 479.745,Z 362.543,A -85,B 0,C 180,E1 -7129.782,E2 -7129.782} C_VEL
LIN {X 0,Y 480.296,Z 347.86,A -85,B 0,C 180,E1 -7130.409,E2 -7130.409} C_VEL
LIN {X 0,Y 480.743,Z 333.334,A -85,B 0,C 180,E1 -7130.86,E2 -7130.86} C_VEL
LIN {X 0,Y 481.136,Z 317.379,A -85,B 0,C 180,E1 -7131.172,E2 -7131.172} C_VEL
LIN {X 0,Y 482.564,Z 182.258,A -85,B 0,C 180,E1 -7133.234,E2 -7133.234} C_VEL
LIN {X 0,Y 478.18,Z 161.558,A -85,B 0,C 180,E1 -7133.814,E2 -7133.814} C_VEL
LIN {X 0,Y 478.42,Z 154.062,A -85,B 0,C 180,E1 -7134.982,E2 -7134.982} C_VEL
LIN {X 0,Y 475.326,Z 140.1,A -85,B 0,C 180,E1 -7137.484,E2 -7137.484} C_VEL
LIN {X 0,Y 474.628,Z 137.199,A -85,B 0,C 180,E1 -7138.051,E2 -7138.051} C_VEL
LIN {X 0,Y 474.575,Z 136.981,A -85,B 0,C 180,E1 -7141.22,E2 -7141.22} C_VEL
LIN {X 0,Y 474.618,Z 136.986,A -85,B 0,C 180,E1 -7144.242,E2 -7144.242} C_VEL
LIN {X 0,Y 474.542,Z 137.001,A -85,B 0,C 180,E1 -7147.388,E2 -7147.388} C_VEL
LIN {X 0,Y 474.6,Z 136.981,A -85,B 0,C 180,E1 -7149.643,E2 -7149.643} C_VEL
LIN {X 0,Y 474.569,Z 136.992,A -85,B 0,C 180,E1 -7152.94,E2 -7152.94} C_VEL
LIN {X 0,Y 474.602,Z 136.987,A -85,B 0,C 180,E1 -7155.894,E2 -7155.894} C_VEL
LIN {X 0,Y 474.591,Z 136.973,A -85,B 0,C 180,E1 -7159.339,E2 -7159.339} C_VEL
LIN {X 0,Y 474.6,Z 136.982,A -85,B 0,C 180,E1 -7161.706,E2 -7161.706} C_VEL
LIN {X 0,Y 474.62,Z 136.987,A -85,B 0,C 180,E1 -7164.725,E2 -7164.725} C_VEL
LIN {X 0,Y 474.628,Z 136.961,A -85,B 0,C 180,E1 -7167.787,E2 -7167.787} C_VEL
LIN {X 0,Y 474.6,Z 136.989,A -85,B 0,C 180,E1 -7170.89,E2 -7170.89} C_VEL
LIN {X 0,Y 474.592,Z 136.989,A -85,B 0,C 180,E1 -7173.624,E2 -7173.624} C_VEL
LIN {X 0,Y 474.636,Z 136.986,A -85,B 0,C 180,E1 -7176.642,E2 -7176.642} C_VEL
LIN {X 0,Y 474.65,Z 136.979,A -85,B 0,C 180,E1 -7180.089,E2 -7180.089} C_VEL
LIN {X 0,Y 474.598,Z 136.989,A -85,B 0,C 180,E1 -7182.772,E2 -7182.772} C_VEL
LIN {X 0,Y 474.638,Z 136.979,A -85,B 0,C 180,E1 -7185.421,E2 -7185.421} C_VEL
LIN {X 0,Y 474.707,Z 136.981,A -85,B 0,C 180,E1 -7188.038,E2 -7188.038} C_VEL
LIN {X 0,Y 474.71,Z 136.97,A -85,B 0,C 180,E1 -7191.486,E2 -7191.486} C_VEL
LIN {X 0,Y 474.76,Z 136.972,A -85,B 0,C 180,E1 -7194.052,E2 -7194.052} C_VEL
LIN {X 0,Y 474.884,Z 136.949,A -85,B 0,C 180,E1 -7197.455,E2 -7197.455} C_VEL
LIN {X 0,Y 474.911,Z 136.951,A -85,B 0,C 180,E1 -7200,E2 -7200} C_VEL
LIN {X 0,Y 474.887,Z 136.947,A -85,B 0,C 180,E1 -7202.545,E2 -7202.545} C_VEL
LIN {X 0,Y 474.762,Z 136.969,A -85,B 0,C 180,E1 -7205.948,E2 -7205.948} C_VEL
LIN {X 0,Y 474.713,Z 136.971,A -85,B 0,C 180,E1 -7208.514,E2 -7208.514} C_VEL
LIN {X 0,Y 474.707,Z 136.975,A -85,B 0,C 180,E1 -7211.962,E2 -7211.962} C_VEL
LIN {X 0,Y 474.701,Z 136.972,A -85,B 0,C 180,E1 -7215.456,E2 -7215.456} C_VEL
LIN {X 0,Y 474.663,Z 136.985,A -85,B 0,C 180,E1 -7219.01,E2 -7219.01} C_VEL
LIN {X 0,Y 474.59,Z 136.986,A -85,B 0,C 180,E1 -7221.729,E2 -7221.729} C_VEL
LIN {X 0,Y 474.631,Z 136.988,A -85,B 0,C 180,E1 -7224.494,E2 -7224.494} C_VEL
LIN {X 0,Y 474.675,Z 136.98,A -85,B 0,C 180,E1 -7227.332,E2 -7227.332} C_VEL
LIN {X 0,Y 474.606,Z 136.988,A -85,B 0,C 180,E1 -7230.23,E2 -7230.23} C_VEL
LIN {X 0,Y 474.615,Z 136.965,A -85,B 0,C 180,E1 -7233.222,E2 -7233.222} C_VEL
LIN {X 0,Y 474.59,Z 136.992,A -85,B 0,C 180,E1 -7236.323,E2 -7236.323} C_VEL
LIN {X 0,Y 474.628,Z 136.976,A -85,B 0,C 180,E1 -7239.647,E2 -7239.647} C_VEL
LIN {X 0,Y 474.615,Z 136.989,A -85,B 0,C 180,E1 -7242.934,E2 -7242.934} C_VEL
LIN {X 0,Y 474.607,Z 136.98,A -85,B 0,C 180,E1 -7245.895,E2 -7245.895} C_VEL
LIN {X 0,Y 474.628,Z 136.985,A -85,B 0,C 180,E1 -7249.041,E2 -7249.041} C_VEL
LIN {X 0,Y 474.611,Z 136.988,A -85,B 0,C 180,E1 -7251.704,E2 -7251.704} C_VEL
LIN {X 0,Y 474.625,Z 136.987,A -85,B 0,C 180,E1 -7254.726,E2 -7254.726} C_VEL
LIN {X 0,Y 474.636,Z 136.961,A -85,B 0,C 180,E1 -7257.788,E2 -7257.788} C_VEL
LIN {X 0,Y 474.672,Z 137.194,A -85,B 0,C 180,E1 -7260.939,E2 -7260.939} C_VEL
LIN {X 0,Y 477.939,Z 150.883,A -85,B 0,C 180,E1 -7263.348,E2 -7263.348} C_VEL
LIN {X 0,Y 478.752,Z 155.398,A -85,B 0,C 180,E1 -7264.105,E2 -7264.105} C_VEL
LIN {X 0,Y 478.059,Z 169.344,A -85,B 0,C 180,E1 -7266.211,E2 -7266.211} C_VEL
LIN {X 0,Y 482.097,Z 189.164,A -85,B 0,C 180,E1 -7266.766,E2 -7266.766} C_VEL
LIN {X 0,Y 482.454,Z 193.723,A -85,B 0,C 180,E1 -7266.856,E2 -7266.856} C_VEL
LIN {X 0,Y 480.891,Z 334.523,A -85,B 0,C 180,E1 -7269.019,E2 -7269.019} C_VEL
LIN {X 0,Y 480.409,Z 350.598,A -85,B 0,C 180,E1 -7269.434,E2 -7269.434} C_VEL
LIN {X 0,Y 479.894,Z 364.529,A -85,B 0,C 180,E1 -7269.96,E2 -7269.96} C_VEL
LIN {X 0,Y 479.214,Z 378.038,A -85,B 0,C 180,E1 -7270.621,E2 -7270.621} C_VEL
LIN {X 0,Y 478.506,Z 390.342,A -85,B 0,C 180,E1 -7271.37,E2 -7271.37} C_VEL
LIN {X 0,Y 477.717,Z 403.351,A -85,B 0,C 180,E1 -7272.336,E2 -7272.336} C_VEL
LIN {X 0,Y 476.914,Z 415.757,A -85,B 0,C 180,E1 -7273.451,E2 -7273.451} C_VEL
LIN {X 0,Y 476.183,Z 426.481,A -85,B 0,C 180,E1 -7274.594,E2 -7274.594} C_VEL
LIN {X 0,Y 475.606,Z 436.709,A -85,B 0,C 180,E1 -7275.888,E2 -7275.888} C_VEL
LIN {X 0,Y 474.913,Z 446.864,A -85,B 0,C 180,E1 -7277.418,E2 -7277.418} C_VEL
LIN {X 0,Y 474.597,Z 455.006,A -85,B 0,C 180,E1 -7278.901,E2 -7278.901} C_VEL
LIN {X 0,Y 474.161,Z 462.8,A -85,B 0,C 180,E1 -7280.616,E2 -7280.616} C_VEL
LIN {X 0,Y 473.941,Z 469,A -85,B 0,C 180,E1 -7282.33,E2 -7282.33} C_VEL
LIN {X 0,Y 473.811,Z 473.794,A -85,B 0,C 180,E1 -7284.04,E2 -7284.04} C_VEL
LIN {X 0,Y 473.686,Z 477.305,A -85,B 0,C 180,E1 -7285.746,E2 -7285.746} C_VEL
LIN {X 0,Y 473.717,Z 479.616,A -85,B 0,C 180,E1 -7287.449,E2 -7287.449} C_VEL
LIN {X 0,Y 473.684,Z 480.778,A -85,B 0,C 180,E1 -7289.15,E2 -7289.15} C_VEL
LIN {X 0,Y 473.684,Z 480.777,A -85,B 0,C 180,E1 -7290.85,E2 -7290.85} C_VEL
LIN {X 0,Y 473.717,Z 479.611,A -85,B 0,C 180,E1 -7292.551,E2 -7292.551} C_VEL
LIN {X 0,Y 473.686,Z 477.3,A -85,B 0,C 180,E1 -7294.254,E2 -7294.254} C_VEL
LIN {X 0,Y 473.833,Z 473.795,A -85,B 0,C 180,E1 -7295.959,E2 -7295.959} C_VEL
LIN {X 0,Y 473.941,Z 469.002,A -85,B 0,C 180,E1 -7297.67,E2 -7297.67} C_VEL
LIN {X 0,Y 474.161,Z 462.794,A -85,B 0,C 180,E1 -7299.383,E2 -7299.383} C_VEL
LIN {X 0,Y 474.6,Z 454.996,A -85,B 0,C 180,E1 -7301.099,E2 -7301.099} C_VEL
LIN {X 0,Y 474.979,Z 446.364,A -85,B 0,C 180,E1 -7302.66,E2 -7302.66} C_VEL
LIN {X 0,Y 475.607,Z 436.702,A -85,B 0,C 180,E1 -7304.112,E2 -7304.112} C_VEL
LIN {X 0,Y 476.205,Z 426.473,A -85,B 0,C 180,E1 -7305.406,E2 -7305.406} C_VEL
LIN {X 0,Y 477.034,Z 413.841,A -85,B 0,C 180,E1 -7306.74,E2 -7306.74} C_VEL
LIN {X 0,Y 477.872,Z 400.715,A -85,B 0,C 180,E1 -7307.879,E2 -7307.879} C_VEL
LIN {X 0,Y 478.692,Z 387.105,A -85,B 0,C 180,E1 -7308.844,E2 -7308.844} C_VEL
LIN {X 0,Y 479.506,Z 373.007,A -85,B 0,C 180,E1 -7309.645,E2 -7309.645} C_VEL
LIN {X 0,Y 480.16,Z 357.657,A -85,B 0,C 180,E1 -7310.318,E2 -7310.318} C_VEL
LIN {X 0,Y 480.684,Z 342.164,A -85,B 0,C 180,E1 -7310.805,E2 -7310.805} C_VEL
LIN {X 0,Y 481.032,Z 326.728,A -85,B 0,C 180,E1 -7311.114,E2 -7311.114} C_VEL
LIN {X 0,Y 482.497,Z 191.569,A -85,B 0,C 180,E1 -7313.173,E2 -7313.173} C_VEL
LIN {X 0,Y 478.039,Z 169.603,A -85,B 0,C 180,E1 -7313.769,E2 -7313.769} C_VEL
LIN {X 0,Y 478.724,Z 155.383,A -85,B 0,C 180,E1 -7315.897,E2 -7315.897} C_VEL
LIN {X 0,Y 476.476,Z 144.519,A -85,B 0,C 180,E1 -7317.749,E2 -7317.749} C_VEL
LIN {X 0,Y 474.634,Z 137.055,A -85,B 0,C 180,E1 -7319.118,E2 -7319.118} C_VEL
LIN {X 0,Y 474.615,Z 136.966,A -85,B 0,C 180,E1 -7322.431,E2 -7322.431} C_VEL
LIN {X 0,Y 474.615,Z 136.987,A -85,B 0,C 180,E1 -7325.469,E2 -7325.469} C_VEL
LIN {X 0,Y 474.612,Z 136.985,A -85,B 0,C 180,E1 -7328.457,E2 -7328.457} C_VEL
LIN {X 0,Y 474.621,Z 136.993,A -85,B 0,C 180,E1 -7331.785,E2 -7331.785} C_VEL
LIN {X 0,Y 474.617,Z 136.981,A -85,B 0,C 180,E1 -7334.702,E2 -7334.702} C_VEL
LIN {X 0,Y 474.625,Z 136.984,A -85,B 0,C 180,E1 -7337.763,E2 -7337.763} C_VEL
LIN {X 0,Y 474.645,Z 136.974,A -85,B 0,C 180,E1 -7340.454,E2 -7340.454} C_VEL
LIN {X 0,Y 474.589,Z 136.992,A -85,B 0,C 180,E1 -7343.677,E2 -7343.677} C_VEL
LIN {X 0,Y 474.615,Z 136.964,A -85,B 0,C 180,E1 -7346.778,E2 -7346.778} C_VEL
LIN {X 0,Y 474.606,Z 136.989,A -85,B 0,C 180,E1 -7349.77,E2 -7349.77} C_VEL
LIN {X 0,Y 474.698,Z 136.977,A -85,B 0,C 180,E1 -7352.68,E2 -7352.68} C_VEL
LIN {X 0,Y 474.656,Z 136.985,A -85,B 0,C 180,E1 -7355.507,E2 -7355.507} C_VEL
LIN {X 0,Y 474.672,Z 136.978,A -85,B 0,C 180,E1 -7359.186,E2 -7359.186} C_VEL
LIN {X 0,Y 474.645,Z 136.983,A -85,B 0,C 180,E1 -7361.884,E2 -7361.884} C_VEL
LIN {X 0,Y 474.701,Z 136.971,A -85,B 0,C 180,E1 -7364.544,E2 -7364.544} C_VEL
LIN {X 0,Y 474.706,Z 136.975,A -85,B 0,C 180,E1 -7368.038,E2 -7368.038} C_VEL
LIN {X 0,Y 474.713,Z 136.971,A -85,B 0,C 180,E1 -7371.486,E2 -7371.486} C_VEL
LIN {X 0,Y 474.747,Z 136.967,A -85,B 0,C 180,E1 -7374.904,E2 -7374.904} C_VEL
LIN {X 0,Y 474.888,Z 136.947,A -85,B 0,C 180,E1 -7377.455,E2 -7377.455} C_VEL
LIN {X 0,Y 474.912,Z 136.95,A -85,B 0,C 180,E1 -7380,E2 -7380} C_VEL
LIN {X 0,Y 474.884,Z 136.948,A -85,B 0,C 180,E1 -7382.545,E2 -7382.545} C_VEL
LIN {X 0,Y 474.76,Z 136.971,A -85,B 0,C 180,E1 -7385.948,E2 -7385.948} C_VEL
LIN {X 0,Y 474.713,Z 136.97,A -85,B 0,C 180,E1 -7388.514,E2 -7388.514} C_VEL
LIN {X 0,Y 474.706,Z 136.98,A -85,B 0,C 180,E1 -7391.962,E2 -7391.962} C_VEL
LIN {X 0,Y 474.69,Z 136.972,A -85,B 0,C 180,E1 -7395.456,E2 -7395.456} C_VEL
LIN {X 0,Y 474.662,Z 136.977,A -85,B 0,C 180,E1 -7399.01,E2 -7399.01} C_VEL
LIN {X 0,Y 474.589,Z 136.991,A -85,B 0,C 180,E1 -7401.729,E2 -7401.729} C_VEL
LIN {X 0,Y 474.627,Z 136.98,A -85,B 0,C 180,E1 -7404.495,E2 -7404.495} C_VEL
